// TIA Portal V18 program export: 0 tag tables, 0 data types, 83 data blocks, 120 code blocks (in call order from the OBs), 84 instance data blocks

DATA_BLOCK "GeneralDebug"   // DB1
{ S7_Optimized_Access := 'TRUE' }
// stored: MemoryReserve 100
   VAR
      Debug : Array[1..99] of Bool;
   END_VAR
BEGIN
END_DATA_BLOCK

DATA_BLOCK "DB_Commissioning"   // DB32767
{ S7_Optimized_Access := 'TRUE' }
// stored: AutoNumber false, MemoryReserve 100
   VAR RETAIN
      str : Array[1..8] of String[60];
      bit : Array[1..8] of Bool;
   END_VAR
BEGIN
   str[1] := 'LE4B171420124M33700000131950710';
END_DATA_BLOCK

DATA_BLOCK "DB_MES_Monitoring"   // DB8
{ S7_Optimized_Access := 'TRUE' }
AUTHOR : caisik - mr. machinist
// stored: MemoryReserve 100
   VAR
      Diag { S7_SetPoint := 'True'} : "UDT_MES_Monitoring";
   END_VAR
BEGIN
END_DATA_BLOCK

DATA_BLOCK "DB_ALL_PROCESS_PARAMETERS"   // DB5000
{ S7_Optimized_Access := 'TRUE' }
// stored: AutoNumber false, MemoryReserve 1000
   VAR RETAIN
      "Choosen Recipe Number" : Bool;
      ACTUAL_CHOOSEN_TYPE : "UDT_OP10_Recipe_type";   // THERE IS ASCTUAL DATA READED OUT FROM LIBRARY OF 20 TYPES BELOW
      PRODUCT_TYPE : Array[1..10] of "UDT_OP10_Recipe_type";   // PACK OF TWENTY DIFFERENT TYPES PRODUCT AND THEIR PARAMETERS FOR THE PROCESS
   END_VAR
BEGIN
   ACTUAL_CHOOSEN_TYPE.Header.RecipeName := 'produkt 1';
   ACTUAL_CHOOSEN_TYPE.Header.RecipeID := 2;
   ACTUAL_CHOOSEN_TYPE.Header."Version" := 19629;
   ACTUAL_CHOOSEN_TYPE.Header.LastModified := DTL#2026-01-17-04:23:27.501;
   ACTUAL_CHOOSEN_TYPE.Header.PartType := 'additional  name';
   ACTUAL_CHOOSEN_TYPE.Process.Timers.Delay_glue_init_start := T#2S;
   ACTUAL_CHOOSEN_TYPE.Process.Timers.Delay_Medium := T#600MS;
   ACTUAL_CHOOSEN_TYPE.Process.Timers.Delay_Long := T#2S;
   ACTUAL_CHOOSEN_TYPE.Process.Timers.Cylinder_ActTime := T#6S;
   ACTUAL_CHOOSEN_TYPE.Process.Limits.RetryLimit := 3;
   ACTUAL_CHOOSEN_TYPE.Process.Press.B1_Program := 1;
   ACTUAL_CHOOSEN_TYPE.Process.Press.B2_Program := 1;
   ACTUAL_CHOOSEN_TYPE.Process.Vision.CGlueShaftIV3_Progs[1] := 16#0001;
   ACTUAL_CHOOSEN_TYPE.Process.Vision.CGlueShaftIV3_Progs[2] := 16#0002;
   ACTUAL_CHOOSEN_TYPE.Process.Vision.CGlueShaftIV3_Progs[3] := 16#0003;
   ACTUAL_CHOOSEN_TYPE.Process.Vision.CGlueShaftIV3_Progs[4] := 16#0004;
   ACTUAL_CHOOSEN_TYPE.Process.Vision.CGlueMagnetIV3_Prog := 16#0001;
   ACTUAL_CHOOSEN_TYPE.Process.Vision.CGlueProgram := 1;
   ACTUAL_CHOOSEN_TYPE."Tooling Code".A1_Table[1] := 'SZ23055-OP010-E-Compressor-ring1 Loading tooling-1';
   ACTUAL_CHOOSEN_TYPE."Tooling Code".A1_Table[2] := 'SZ23055-OP010-E-Compressor-ring1 Loading tooling-2';
   ACTUAL_CHOOSEN_TYPE."Tooling Code".A1_Table[3] := 'SZ23055-OP010-E-Compressor-ring1 Loading tooling-3';
   ACTUAL_CHOOSEN_TYPE."Tooling Code".A1_Table[4] := 'SZ23055-OP010-E-Compressor-ring1 Loading tooling-4';
   ACTUAL_CHOOSEN_TYPE."Tooling Code".A1_Table[5] := 'SZ23055-OP010-E-Compressor-ring1 Loading tooling-5';
   ACTUAL_CHOOSEN_TYPE."Tooling Code".A1_Table[6] := 'SZ23055-OP010-E-Compressor-ring1 Loading tooling-6';
   ACTUAL_CHOOSEN_TYPE."Tooling Code".A1_Table[7] := 'SZ23055-OP010-E-Compressor-ring1 Loading tooling-7';
   ACTUAL_CHOOSEN_TYPE."Tooling Code".A1_Table[8] := 'SZ23055-OP010-E-Compressor-ring1 Loading tooling-8';
   ACTUAL_CHOOSEN_TYPE."Tooling Code".A2_Table[1] := 'SZ23055-OP010-E-Compresspr-ring1 cutting tool';
   ACTUAL_CHOOSEN_TYPE."Tooling Code".A2_Table[2] := 'SZ23055-OP010-E-Compressor-Left NG tooling-1';
   ACTUAL_CHOOSEN_TYPE."Tooling Code".A2_Table[3] := 'SZ23055-OP010-E-Compressor-shaft Rotating scanning tooling-1';
   ACTUAL_CHOOSEN_TYPE."Tooling Code".A2_Table[4] := 'SZ23055-OP010-E-Compressor-ring1 Below Positioning fixture -1';
   ACTUAL_CHOOSEN_TYPE."Tooling Code".A2_Table[5] := 'SZ23055-OP010-E-Compressor-Point adhesive tooling-1';
   ACTUAL_CHOOSEN_TYPE."Tooling Code".A2_Table[6] := 'SZ23055-OP010-E-Compressor-ring1 Upper pressing fixture-1';
   ACTUAL_CHOOSEN_TYPE."Tooling Code".A2_Table[7] := 'SZ23055-OP010-E-Compresspr-ring2 cutting tool';
   ACTUAL_CHOOSEN_TYPE."Tooling Code".A2_Table[8] := 'SZ23055-OP010-E-Compressor-Right NG tooling-1';
   ACTUAL_CHOOSEN_TYPE."Tooling Code".ROB1_Shaft_Handling_Robot.Gripper."JAW TOOLING LEFT" := 'SZ23055-OP010-E-Compressor-robot1 ring1 Left clamping jaw tooling-1';
   ACTUAL_CHOOSEN_TYPE."Tooling Code".ROB1_Shaft_Handling_Robot.Gripper."JAW TOOLING RIGHT" := 'SZ23055-OP010-E-Compressor-robot1 ring1 Right clamping jaw tooling-2';
   ACTUAL_CHOOSEN_TYPE."Tooling Code".ROB1_Shaft_Handling_Robot.Gripper."SHAFT CLAMPING LEFT" := 'SZ23055-OP010-E-Compressor-robot1 shaft Left clamping jaw tooling-1';
   ACTUAL_CHOOSEN_TYPE."Tooling Code".ROB1_Shaft_Handling_Robot.Gripper."SHAFT CLAMPING RIGHT" := 'SZ23055-OP010-E-Compressor-robot1 shaft Right clamping jaw tooling-2';
   ACTUAL_CHOOSEN_TYPE."Tooling Code".ROB2_Main_Assembly_Robot.Gripper."JAW TOOLING LEFT" := 'SZ23055-OP010-E-Compressor-robot2 shaft Right clamping jaw tooling-2';
   ACTUAL_CHOOSEN_TYPE."Tooling Code".ROB2_Main_Assembly_Robot.Gripper."JAW TOOLING RIGHT" := 'SZ23055-OP010-E-Compressor-robot2 shaft Left clamping jaw tooling-1';
   ACTUAL_CHOOSEN_TYPE."Tooling Code".ROB2_Main_Assembly_Robot.Gripper."SHAFT CLAMPING LEFT" := 'SZ23055-OP010-E-Compressor-robot2 magnet Right clamping jaw tooling-2';
   ACTUAL_CHOOSEN_TYPE."Tooling Code".ROB2_Main_Assembly_Robot.Gripper."SHAFT CLAMPING RIGHT" := 'SZ23055-OP010-E-Compressor-robot2 magnet Right clamping jaw tooling-2';
   ACTUAL_CHOOSEN_TYPE."Tooling Code".ROB3_Unloading_Robot.Gripper."JAW TOOLING LEFT" := 'SZ23055-OP010-E-Compressor-robot3 ring2 Right clamping jaw tooling-2';
   ACTUAL_CHOOSEN_TYPE."Tooling Code".ROB3_Unloading_Robot.Gripper."JAW TOOLING RIGHT" := 'SZ23055-OP010-E-Compressor-robot3 ring2 Left clamping jaw tooling-1';
   ACTUAL_CHOOSEN_TYPE."Tooling Code".ROB3_Unloading_Robot.Gripper."SHAFT CLAMPING LEFT" := 'SZ23055-OP010-E-Compressor-robot3 shaft Left clamping jaw tooling-1';
   ACTUAL_CHOOSEN_TYPE."Tooling Code".ROB3_Unloading_Robot.Gripper."SHAFT CLAMPING RIGHT" := 'SZ23055-OP010-E-Compressor-robot3 shaft Right clamping jaw tooling-2';
   ACTUAL_CHOOSEN_TYPE."Tooling Code".A1_Fixtures.A1RingUnloadingFixtureCode := 'SZ23055-OP010-E-Compresspr-ring1 cutting tool';
   ACTUAL_CHOOSEN_TYPE."Tooling Code".A1_Fixtures.E1LoadingNGFixtureCode := 'SZ23055-OP010-E-Compressor-Left NG tooling-1';
   ACTUAL_CHOOSEN_TYPE."Tooling Code".A1_Fixtures.ShaftScanFixtureCode := 'SZ23055-OP010-E-Compressor-shaft Rotating scanning tooling-1';
   ACTUAL_CHOOSEN_TYPE."Tooling Code".A1_Fixtures.B1PressFixtureCode := 'SZ23055-OP010-E-Compressor-ring1 Below Positioning fixture -1';
   ACTUAL_CHOOSEN_TYPE."Tooling Code".A1_Fixtures.CGlueFixtureCode := 'SZ23055-OP010-E-Compressor-Point adhesive tooling-1';
   ACTUAL_CHOOSEN_TYPE."Tooling Code".A1_Fixtures.B1PressCylFixtureCode := 'SZ23055-OP010-E-Compressor-ring1 Upper pressing fixture-1';
   ACTUAL_CHOOSEN_TYPE."Tooling Code".A2_Fixtures.A2RingUnloadingFixtureCode := 'SZ23055-OP010-E-Compresspr-ring2 cutting tool';
   ACTUAL_CHOOSEN_TYPE."Tooling Code".A2_Fixtures.E2UnloadingNGFixtureCode := 'SZ23055-OP010-E-Compressor-Right NG tooling-1';
   ACTUAL_CHOOSEN_TYPE."Tooling Code".A2_Fixtures.B2PressFixtureCode := 'SZ23055-OP010-E-Compressor-ring2 Below Positioning fixture -1';
   ACTUAL_CHOOSEN_TYPE."Tooling Code".A2_Fixtures.CGlueNGFixtureCode := 'SZ23055-OP010-E-Compressor-NG middle shift tooling-1';
   ACTUAL_CHOOSEN_TYPE."Tooling Code".A2_Fixtures.B2PressCylFixtureCode := 'SZ23055-OP010-E-Compressor-ring2 Upper pressing fixture-1';
   ACTUAL_CHOOSEN_TYPE.Motion.Gluing_Nozzle_Z.Position[1].Pos := 143.76;
   ACTUAL_CHOOSEN_TYPE.Motion.Gluing_Nozzle_Z.Position[2].Pos := 139.11;
   ACTUAL_CHOOSEN_TYPE.Motion.Gluing_Nozzle_Z.Position[3].Pos := 131.98;
   ACTUAL_CHOOSEN_TYPE.Motion.Gluing_Nozzle_Z.Position[4].Pos := 127.89;
   ACTUAL_CHOOSEN_TYPE.Motion.Gluing_Nozzle_Z.Position[6].Pos := 127.0;
   ACTUAL_CHOOSEN_TYPE.Motion.Gluing_Nozzle_Z.Position[7].Pos := 48.11;
   ACTUAL_CHOOSEN_TYPE.Motion.Gluing_Nozzle_Z.Position[9].Pos := 123.0;
   ACTUAL_CHOOSEN_TYPE.Motion.Gluing_Nozzle_Z.Position[1..4].Vel := 200;
   ACTUAL_CHOOSEN_TYPE.Motion.Gluing_Nozzle_Z.Position[6..9].Vel := 200;
   ACTUAL_CHOOSEN_TYPE.Motion.Gluing_Nozzle_X.Position[1].Pos := 2.34;
   ACTUAL_CHOOSEN_TYPE.Motion.Gluing_Nozzle_X.Position[2].Pos := 76.0;
   ACTUAL_CHOOSEN_TYPE.Motion.Gluing_Nozzle_X.Position[3..6].Pos := 84.69;
   ACTUAL_CHOOSEN_TYPE.Motion.Gluing_Nozzle_X.Position[7].Pos := 85.0;
   ACTUAL_CHOOSEN_TYPE.Motion.Gluing_Nozzle_X.Position[8].Pos := 88.53;
   ACTUAL_CHOOSEN_TYPE.Motion.Gluing_Nozzle_X.Position[1..8].Vel := 200;
   ACTUAL_CHOOSEN_TYPE.Motion.Gluing_Nozzle_Y.Position[1..5].Pos := 115.47;
   ACTUAL_CHOOSEN_TYPE.Motion.Gluing_Nozzle_Y.Position[6].Pos := 110.18;
   ACTUAL_CHOOSEN_TYPE.Motion.Gluing_Nozzle_Y.Position[7].Pos := 60.52;
   ACTUAL_CHOOSEN_TYPE.Motion.Gluing_Nozzle_Y.Position[8].Pos := 80.0;
   ACTUAL_CHOOSEN_TYPE.Motion.Gluing_Nozzle_Y.Position[1..7].Vel := 200;
   ACTUAL_CHOOSEN_TYPE.Motion.Gluing_Nozzle_Y.Position[8].Vel := 100;
   ACTUAL_CHOOSEN_TYPE.Motion.Ring_Turntable_Axis_1.Position[1].Pos := 3419;
   ACTUAL_CHOOSEN_TYPE.Motion.Ring_Turntable_Axis_1.Position[2].Pos := 48386;
   ACTUAL_CHOOSEN_TYPE.Motion.Ring_Turntable_Axis_1.Position[3].Pos := 93294;
   ACTUAL_CHOOSEN_TYPE.Motion.Ring_Turntable_Axis_1.Position[4].Pos := 138335;
   ACTUAL_CHOOSEN_TYPE.Motion.Ring_Turntable_Axis_1.Position[5].Pos := 183464;
   ACTUAL_CHOOSEN_TYPE.Motion.Ring_Turntable_Axis_1.Position[6].Pos := 228443;
   ACTUAL_CHOOSEN_TYPE.Motion.Ring_Turntable_Axis_1.Position[7].Pos := 273535;
   ACTUAL_CHOOSEN_TYPE.Motion.Ring_Turntable_Axis_1.Position[8].Pos := 318250;
   ACTUAL_CHOOSEN_TYPE.Motion.Ring_Turntable_Axis_1.Position[1..8].Vel := 10000;
   ACTUAL_CHOOSEN_TYPE.Motion.Shaft_Scan_Turntable_Axis.Position[2].Pos := 450000;
   ACTUAL_CHOOSEN_TYPE.Motion.Shaft_Scan_Turntable_Axis.Position[3].Pos := 900000;
   ACTUAL_CHOOSEN_TYPE.Motion.Shaft_Scan_Turntable_Axis.Position[4].Pos := 135000;
   ACTUAL_CHOOSEN_TYPE.Motion.Shaft_Scan_Turntable_Axis.Position[5].Pos := 180000;
   ACTUAL_CHOOSEN_TYPE.Motion.Shaft_Scan_Turntable_Axis.Position[6].Pos := 225000;
   ACTUAL_CHOOSEN_TYPE.Motion.Shaft_Scan_Turntable_Axis.Position[7].Pos := 270000;
   ACTUAL_CHOOSEN_TYPE.Motion.Shaft_Scan_Turntable_Axis.Position[8].Pos := 315000;
   ACTUAL_CHOOSEN_TYPE.Motion.Shaft_Scan_Turntable_Axis.Position[1..8].Vel := 10000;
   ACTUAL_CHOOSEN_TYPE.Motion.Gluing_Rotary_Jig_Axis.Position[3..6].Pos := 680000;
   ACTUAL_CHOOSEN_TYPE.Motion.Gluing_Rotary_Jig_Axis.Position[7].Pos := 90000;
   ACTUAL_CHOOSEN_TYPE.Motion.Gluing_Rotary_Jig_Axis.Position[8].Pos := 180000;
   ACTUAL_CHOOSEN_TYPE.Motion.Gluing_Rotary_Jig_Axis.Position[9].Pos := 270000;
   ACTUAL_CHOOSEN_TYPE.Motion.Gluing_Rotary_Jig_Axis.Position[1..2].Vel := 20000;
   ACTUAL_CHOOSEN_TYPE.Motion.Gluing_Rotary_Jig_Axis.Position[3..9].Vel := 10000;
   ACTUAL_CHOOSEN_TYPE.Motion.Ring_Turntable_Axis_2.Position[1].Pos := 3585;
   ACTUAL_CHOOSEN_TYPE.Motion.Ring_Turntable_Axis_2.Position[2].Pos := 48610;
   ACTUAL_CHOOSEN_TYPE.Motion.Ring_Turntable_Axis_2.Position[3].Pos := 93637;
   ACTUAL_CHOOSEN_TYPE.Motion.Ring_Turntable_Axis_2.Position[4].Pos := 138606;
   ACTUAL_CHOOSEN_TYPE.Motion.Ring_Turntable_Axis_2.Position[5].Pos := 183388;
   ACTUAL_CHOOSEN_TYPE.Motion.Ring_Turntable_Axis_2.Position[6].Pos := 228458;
   ACTUAL_CHOOSEN_TYPE.Motion.Ring_Turntable_Axis_2.Position[7].Pos := 273513;
   ACTUAL_CHOOSEN_TYPE.Motion.Ring_Turntable_Axis_2.Position[8].Pos := 318501;
   ACTUAL_CHOOSEN_TYPE.Motion.Ring_Turntable_Axis_2.Position[1..8].Vel := 10000;
   PRODUCT_TYPE[1].Header.RecipeName := 'produkt 1';
   PRODUCT_TYPE[3].Header.RecipeName := 'produkt 1';
   PRODUCT_TYPE[10].Header.RecipeName := 'produkt 1';
   PRODUCT_TYPE[1].Header.RecipeID := 1;
   PRODUCT_TYPE[3].Header.RecipeID := 1;
   PRODUCT_TYPE[10].Header.RecipeID := 1;
   PRODUCT_TYPE[1].Header."Version" := 1;
   PRODUCT_TYPE[3].Header."Version" := 1;
   PRODUCT_TYPE[10].Header."Version" := 1;
   PRODUCT_TYPE[1].Header.LastModified := DTL#2026-01-17-04:23:27.501;
   PRODUCT_TYPE[3].Header.LastModified := DTL#2026-01-17-04:23:27.501;
   PRODUCT_TYPE[10].Header.LastModified := DTL#2026-01-17-04:23:27.501;
   PRODUCT_TYPE[1].Header.PartType := 'additional  name';
   PRODUCT_TYPE[3].Header.PartType := 'additional  name';
   PRODUCT_TYPE[10].Header.PartType := 'additional  name';
   PRODUCT_TYPE[1].Process.Timers.Delay_glue_init_start := T#2S;
   PRODUCT_TYPE[2].Process.Timers.Delay_glue_init_start := T#0MS;
   PRODUCT_TYPE[3].Process.Timers.Delay_glue_init_start := T#300MS;
   PRODUCT_TYPE[4..9].Process.Timers.Delay_glue_init_start := T#0MS;
   PRODUCT_TYPE[10].Process.Timers.Delay_glue_init_start := T#2S;
   PRODUCT_TYPE[1].Process.Timers.Delay_Medium := T#600MS;
   PRODUCT_TYPE[3].Process.Timers.Delay_Medium := T#600MS;
   PRODUCT_TYPE[10].Process.Timers.Delay_Medium := T#600MS;
   PRODUCT_TYPE[1].Process.Timers.Delay_Long := T#2S;
   PRODUCT_TYPE[3].Process.Timers.Delay_Long := T#2S;
   PRODUCT_TYPE[10].Process.Timers.Delay_Long := T#2S;
   PRODUCT_TYPE[1].Process.Timers.Cylinder_ActTime := T#6S;
   PRODUCT_TYPE[3].Process.Timers.Cylinder_ActTime := T#6S;
   PRODUCT_TYPE[10].Process.Timers.Cylinder_ActTime := T#6S;
   PRODUCT_TYPE[1].Process.Limits.RetryLimit := 3;
   PRODUCT_TYPE[3].Process.Limits.RetryLimit := 3;
   PRODUCT_TYPE[10].Process.Limits.RetryLimit := 3;
   PRODUCT_TYPE[1].Process.Press.B1_Program := 1;
   PRODUCT_TYPE[3].Process.Press.B1_Program := 1;
   PRODUCT_TYPE[10].Process.Press.B1_Program := 1;
   PRODUCT_TYPE[1].Process.Press.B2_Program := 1;
   PRODUCT_TYPE[3].Process.Press.B2_Program := 1;
   PRODUCT_TYPE[10].Process.Press.B2_Program := 1;
   PRODUCT_TYPE[1].Process.Vision.CGlueShaftIV3_Progs[1] := 16#0001;
   PRODUCT_TYPE[1].Process.Vision.CGlueShaftIV3_Progs[2] := 16#0002;
   PRODUCT_TYPE[1].Process.Vision.CGlueShaftIV3_Progs[3] := 16#0003;
   PRODUCT_TYPE[1].Process.Vision.CGlueShaftIV3_Progs[4] := 16#0004;
   PRODUCT_TYPE[3].Process.Vision.CGlueShaftIV3_Progs[1] := 16#0001;
   PRODUCT_TYPE[3].Process.Vision.CGlueShaftIV3_Progs[2] := 16#0002;
   PRODUCT_TYPE[3].Process.Vision.CGlueShaftIV3_Progs[3] := 16#0003;
   PRODUCT_TYPE[3].Process.Vision.CGlueShaftIV3_Progs[4] := 16#0004;
   PRODUCT_TYPE[10].Process.Vision.CGlueShaftIV3_Progs[1] := 16#0001;
   PRODUCT_TYPE[10].Process.Vision.CGlueShaftIV3_Progs[2] := 16#0002;
   PRODUCT_TYPE[10].Process.Vision.CGlueShaftIV3_Progs[3] := 16#0003;
   PRODUCT_TYPE[10].Process.Vision.CGlueShaftIV3_Progs[4] := 16#0004;
   PRODUCT_TYPE[1].Process.Vision.CGlueMagnetIV3_Prog := 16#0001;
   PRODUCT_TYPE[3].Process.Vision.CGlueMagnetIV3_Prog := 16#0001;
   PRODUCT_TYPE[10].Process.Vision.CGlueMagnetIV3_Prog := 16#0001;
   PRODUCT_TYPE[1].Process.Vision.CGlueProgram := 1;
   PRODUCT_TYPE[3].Process.Vision.CGlueProgram := 1;
   PRODUCT_TYPE[10].Process.Vision.CGlueProgram := 1;
   PRODUCT_TYPE[1]."Tooling Code".A1_Table[1] := 'SZ23055-OP010-E-Compressor-ring1 Loading tooling-1';
   PRODUCT_TYPE[1]."Tooling Code".A1_Table[2] := 'SZ23055-OP010-E-Compressor-ring1 Loading tooling-2';
   PRODUCT_TYPE[1]."Tooling Code".A1_Table[3] := 'SZ23055-OP010-E-Compressor-ring1 Loading tooling-3';
   PRODUCT_TYPE[1]."Tooling Code".A1_Table[4] := 'SZ23055-OP010-E-Compressor-ring1 Loading tooling-4';
   PRODUCT_TYPE[1]."Tooling Code".A1_Table[5] := 'SZ23055-OP010-E-Compressor-ring1 Loading tooling-5';
   PRODUCT_TYPE[1]."Tooling Code".A1_Table[6] := 'SZ23055-OP010-E-Compressor-ring1 Loading tooling-6';
   PRODUCT_TYPE[1]."Tooling Code".A1_Table[7] := 'SZ23055-OP010-E-Compressor-ring1 Loading tooling-7';
   PRODUCT_TYPE[1]."Tooling Code".A1_Table[8] := 'SZ23055-OP010-E-Compressor-ring1 Loading tooling-8';
   PRODUCT_TYPE[3]."Tooling Code".A1_Table[1] := 'SZ23055-OP010-E-Compressor-ring1 Loading tooling-1';
   PRODUCT_TYPE[3]."Tooling Code".A1_Table[2] := 'SZ23055-OP010-E-Compressor-ring1 Loading tooling-2';
   PRODUCT_TYPE[3]."Tooling Code".A1_Table[3] := 'SZ23055-OP010-E-Compressor-ring1 Loading tooling-3';
   PRODUCT_TYPE[3]."Tooling Code".A1_Table[4] := 'SZ23055-OP010-E-Compressor-ring1 Loading tooling-4';
   PRODUCT_TYPE[3]."Tooling Code".A1_Table[5] := 'SZ23055-OP010-E-Compressor-ring1 Loading tooling-5';
   PRODUCT_TYPE[3]."Tooling Code".A1_Table[6] := 'SZ23055-OP010-E-Compressor-ring1 Loading tooling-6';
   PRODUCT_TYPE[3]."Tooling Code".A1_Table[7] := 'SZ23055-OP010-E-Compressor-ring1 Loading tooling-7';
   PRODUCT_TYPE[3]."Tooling Code".A1_Table[8] := 'SZ23055-OP010-E-Compressor-ring1 Loading tooling-8';
   PRODUCT_TYPE[10]."Tooling Code".A1_Table[1] := 'SZ23055-OP010-E-Compressor-ring1 Loading tooling-1';
   PRODUCT_TYPE[10]."Tooling Code".A1_Table[2] := 'SZ23055-OP010-E-Compressor-ring1 Loading tooling-2';
   PRODUCT_TYPE[10]."Tooling Code".A1_Table[3] := 'SZ23055-OP010-E-Compressor-ring1 Loading tooling-3';
   PRODUCT_TYPE[10]."Tooling Code".A1_Table[4] := 'SZ23055-OP010-E-Compressor-ring1 Loading tooling-4';
   PRODUCT_TYPE[10]."Tooling Code".A1_Table[5] := 'SZ23055-OP010-E-Compressor-ring1 Loading tooling-5';
   PRODUCT_TYPE[10]."Tooling Code".A1_Table[6] := 'SZ23055-OP010-E-Compressor-ring1 Loading tooling-6';
   PRODUCT_TYPE[10]."Tooling Code".A1_Table[7] := 'SZ23055-OP010-E-Compressor-ring1 Loading tooling-7';
   PRODUCT_TYPE[10]."Tooling Code".A1_Table[8] := 'SZ23055-OP010-E-Compressor-ring1 Loading tooling-8';
   PRODUCT_TYPE[1]."Tooling Code".A2_Table[1] := 'SZ23055-OP010-E-Compresspr-ring1 cutting tool';
   PRODUCT_TYPE[1]."Tooling Code".A2_Table[2] := 'SZ23055-OP010-E-Compressor-Left NG tooling-1';
   PRODUCT_TYPE[1]."Tooling Code".A2_Table[3] := 'SZ23055-OP010-E-Compressor-shaft Rotating scanning tooling-1';
   PRODUCT_TYPE[1]."Tooling Code".A2_Table[4] := 'SZ23055-OP010-E-Compressor-ring1 Below Positioning fixture -1';
   PRODUCT_TYPE[1]."Tooling Code".A2_Table[5] := 'SZ23055-OP010-E-Compressor-Point adhesive tooling-1';
   PRODUCT_TYPE[1]."Tooling Code".A2_Table[6] := 'SZ23055-OP010-E-Compressor-ring1 Upper pressing fixture-1';
   PRODUCT_TYPE[1]."Tooling Code".A2_Table[7] := 'SZ23055-OP010-E-Compresspr-ring2 cutting tool';
   PRODUCT_TYPE[1]."Tooling Code".A2_Table[8] := 'SZ23055-OP010-E-Compressor-Right NG tooling-1';
   PRODUCT_TYPE[3]."Tooling Code".A2_Table[1] := 'SZ23055-OP010-E-Compresspr-ring1 cutting tool';
   PRODUCT_TYPE[3]."Tooling Code".A2_Table[2] := 'SZ23055-OP010-E-Compressor-Left NG tooling-1';
   PRODUCT_TYPE[3]."Tooling Code".A2_Table[3] := 'SZ23055-OP010-E-Compressor-shaft Rotating scanning tooling-1';
   PRODUCT_TYPE[3]."Tooling Code".A2_Table[4] := 'SZ23055-OP010-E-Compressor-ring1 Below Positioning fixture -1';
   PRODUCT_TYPE[3]."Tooling Code".A2_Table[5] := 'SZ23055-OP010-E-Compressor-Point adhesive tooling-1';
   PRODUCT_TYPE[3]."Tooling Code".A2_Table[6] := 'SZ23055-OP010-E-Compressor-ring1 Upper pressing fixture-1';
   PRODUCT_TYPE[3]."Tooling Code".A2_Table[7] := 'SZ23055-OP010-E-Compresspr-ring2 cutting tool';
   PRODUCT_TYPE[3]."Tooling Code".A2_Table[8] := 'SZ23055-OP010-E-Compressor-Right NG tooling-1';
   PRODUCT_TYPE[10]."Tooling Code".A2_Table[1] := 'SZ23055-OP010-E-Compresspr-ring1 cutting tool';
   PRODUCT_TYPE[10]."Tooling Code".A2_Table[2] := 'SZ23055-OP010-E-Compressor-Left NG tooling-1';
   PRODUCT_TYPE[10]."Tooling Code".A2_Table[3] := 'SZ23055-OP010-E-Compressor-shaft Rotating scanning tooling-1';
   PRODUCT_TYPE[10]."Tooling Code".A2_Table[4] := 'SZ23055-OP010-E-Compressor-ring1 Below Positioning fixture -1';
   PRODUCT_TYPE[10]."Tooling Code".A2_Table[5] := 'SZ23055-OP010-E-Compressor-Point adhesive tooling-1';
   PRODUCT_TYPE[10]."Tooling Code".A2_Table[6] := 'SZ23055-OP010-E-Compressor-ring1 Upper pressing fixture-1';
   PRODUCT_TYPE[10]."Tooling Code".A2_Table[7] := 'SZ23055-OP010-E-Compresspr-ring2 cutting tool';
   PRODUCT_TYPE[10]."Tooling Code".A2_Table[8] := 'SZ23055-OP010-E-Compressor-Right NG tooling-1';
   PRODUCT_TYPE[1]."Tooling Code".ROB1_Shaft_Handling_Robot.Gripper."JAW TOOLING LEFT" := 'SZ23055-OP010-E-Compressor-robot1 ring1 Left clamping jaw tooling-1';
   PRODUCT_TYPE[3]."Tooling Code".ROB1_Shaft_Handling_Robot.Gripper."JAW TOOLING LEFT" := 'SZ23055-OP010-E-Compressor-robot1 ring1 Left clamping jaw tooling-1';
   PRODUCT_TYPE[10]."Tooling Code".ROB1_Shaft_Handling_Robot.Gripper."JAW TOOLING LEFT" := 'SZ23055-OP010-E-Compressor-robot1 ring1 Left clamping jaw tooling-1';
   PRODUCT_TYPE[1]."Tooling Code".ROB1_Shaft_Handling_Robot.Gripper."JAW TOOLING RIGHT" := 'SZ23055-OP010-E-Compressor-robot1 ring1 Right clamping jaw tooling-2';
   PRODUCT_TYPE[3]."Tooling Code".ROB1_Shaft_Handling_Robot.Gripper."JAW TOOLING RIGHT" := 'SZ23055-OP010-E-Compressor-robot1 ring1 Right clamping jaw tooling-2';
   PRODUCT_TYPE[10]."Tooling Code".ROB1_Shaft_Handling_Robot.Gripper."JAW TOOLING RIGHT" := 'SZ23055-OP010-E-Compressor-robot1 ring1 Right clamping jaw tooling-2';
   PRODUCT_TYPE[1]."Tooling Code".ROB1_Shaft_Handling_Robot.Gripper."SHAFT CLAMPING LEFT" := 'SZ23055-OP010-E-Compressor-robot1 shaft Left clamping jaw tooling-1';
   PRODUCT_TYPE[3]."Tooling Code".ROB1_Shaft_Handling_Robot.Gripper."SHAFT CLAMPING LEFT" := 'SZ23055-OP010-E-Compressor-robot1 shaft Left clamping jaw tooling-1';
   PRODUCT_TYPE[10]."Tooling Code".ROB1_Shaft_Handling_Robot.Gripper."SHAFT CLAMPING LEFT" := 'SZ23055-OP010-E-Compressor-robot1 shaft Left clamping jaw tooling-1';
   PRODUCT_TYPE[1]."Tooling Code".ROB1_Shaft_Handling_Robot.Gripper."SHAFT CLAMPING RIGHT" := 'SZ23055-OP010-E-Compressor-robot1 shaft Right clamping jaw tooling-2';
   PRODUCT_TYPE[3]."Tooling Code".ROB1_Shaft_Handling_Robot.Gripper."SHAFT CLAMPING RIGHT" := 'SZ23055-OP010-E-Compressor-robot1 shaft Right clamping jaw tooling-2';
   PRODUCT_TYPE[10]."Tooling Code".ROB1_Shaft_Handling_Robot.Gripper."SHAFT CLAMPING RIGHT" := 'SZ23055-OP010-E-Compressor-robot1 shaft Right clamping jaw tooling-2';
   PRODUCT_TYPE[1]."Tooling Code".ROB2_Main_Assembly_Robot.Gripper."JAW TOOLING LEFT" := 'SZ23055-OP010-E-Compressor-robot2 shaft Right clamping jaw tooling-2';
   PRODUCT_TYPE[3]."Tooling Code".ROB2_Main_Assembly_Robot.Gripper."JAW TOOLING LEFT" := 'SZ23055-OP010-E-Compressor-robot2 shaft Right clamping jaw tooling-2';
   PRODUCT_TYPE[10]."Tooling Code".ROB2_Main_Assembly_Robot.Gripper."JAW TOOLING LEFT" := 'SZ23055-OP010-E-Compressor-robot2 shaft Right clamping jaw tooling-2';
   PRODUCT_TYPE[1]."Tooling Code".ROB2_Main_Assembly_Robot.Gripper."JAW TOOLING RIGHT" := 'SZ23055-OP010-E-Compressor-robot2 shaft Left clamping jaw tooling-1';
   PRODUCT_TYPE[3]."Tooling Code".ROB2_Main_Assembly_Robot.Gripper."JAW TOOLING RIGHT" := 'SZ23055-OP010-E-Compressor-robot2 shaft Left clamping jaw tooling-1';
   PRODUCT_TYPE[10]."Tooling Code".ROB2_Main_Assembly_Robot.Gripper."JAW TOOLING RIGHT" := 'SZ23055-OP010-E-Compressor-robot2 shaft Left clamping jaw tooling-1';
   PRODUCT_TYPE[1]."Tooling Code".ROB2_Main_Assembly_Robot.Gripper."SHAFT CLAMPING LEFT" := 'SZ23055-OP010-E-Compressor-robot2 magnet Right clamping jaw tooling-2';
   PRODUCT_TYPE[3]."Tooling Code".ROB2_Main_Assembly_Robot.Gripper."SHAFT CLAMPING LEFT" := 'SZ23055-OP010-E-Compressor-robot2 magnet Right clamping jaw tooling-2';
   PRODUCT_TYPE[10]."Tooling Code".ROB2_Main_Assembly_Robot.Gripper."SHAFT CLAMPING LEFT" := 'SZ23055-OP010-E-Compressor-robot2 magnet Right clamping jaw tooling-2';
   PRODUCT_TYPE[1]."Tooling Code".ROB2_Main_Assembly_Robot.Gripper."SHAFT CLAMPING RIGHT" := 'SZ23055-OP010-E-Compressor-robot2 magnet Right clamping jaw tooling-2';
   PRODUCT_TYPE[3]."Tooling Code".ROB2_Main_Assembly_Robot.Gripper."SHAFT CLAMPING RIGHT" := 'SZ23055-OP010-E-Compressor-robot2 magnet Right clamping jaw tooling-2';
   PRODUCT_TYPE[10]."Tooling Code".ROB2_Main_Assembly_Robot.Gripper."SHAFT CLAMPING RIGHT" := 'SZ23055-OP010-E-Compressor-robot2 magnet Right clamping jaw tooling-2';
   PRODUCT_TYPE[1]."Tooling Code".ROB3_Unloading_Robot.Gripper."JAW TOOLING LEFT" := 'SZ23055-OP010-E-Compressor-robot3 ring2 Right clamping jaw tooling-2';
   PRODUCT_TYPE[3]."Tooling Code".ROB3_Unloading_Robot.Gripper."JAW TOOLING LEFT" := 'SZ23055-OP010-E-Compressor-robot3 ring2 Right clamping jaw tooling-2';
   PRODUCT_TYPE[10]."Tooling Code".ROB3_Unloading_Robot.Gripper."JAW TOOLING LEFT" := 'SZ23055-OP010-E-Compressor-robot3 ring2 Right clamping jaw tooling-2';
   PRODUCT_TYPE[1]."Tooling Code".ROB3_Unloading_Robot.Gripper."JAW TOOLING RIGHT" := 'SZ23055-OP010-E-Compressor-robot3 ring2 Left clamping jaw tooling-1';
   PRODUCT_TYPE[3]."Tooling Code".ROB3_Unloading_Robot.Gripper."JAW TOOLING RIGHT" := 'SZ23055-OP010-E-Compressor-robot3 ring2 Left clamping jaw tooling-1';
   PRODUCT_TYPE[10]."Tooling Code".ROB3_Unloading_Robot.Gripper."JAW TOOLING RIGHT" := 'SZ23055-OP010-E-Compressor-robot3 ring2 Left clamping jaw tooling-1';
   PRODUCT_TYPE[1]."Tooling Code".ROB3_Unloading_Robot.Gripper."SHAFT CLAMPING LEFT" := 'SZ23055-OP010-E-Compressor-robot3 shaft Left clamping jaw tooling-1';
   PRODUCT_TYPE[3]."Tooling Code".ROB3_Unloading_Robot.Gripper."SHAFT CLAMPING LEFT" := 'SZ23055-OP010-E-Compressor-robot3 shaft Left clamping jaw tooling-1';
   PRODUCT_TYPE[10]."Tooling Code".ROB3_Unloading_Robot.Gripper."SHAFT CLAMPING LEFT" := 'SZ23055-OP010-E-Compressor-robot3 shaft Left clamping jaw tooling-1';
   PRODUCT_TYPE[1]."Tooling Code".ROB3_Unloading_Robot.Gripper."SHAFT CLAMPING RIGHT" := 'SZ23055-OP010-E-Compressor-robot3 shaft Right clamping jaw tooling-2';
   PRODUCT_TYPE[3]."Tooling Code".ROB3_Unloading_Robot.Gripper."SHAFT CLAMPING RIGHT" := 'SZ23055-OP010-E-Compressor-robot3 shaft Right clamping jaw tooling-2';
   PRODUCT_TYPE[10]."Tooling Code".ROB3_Unloading_Robot.Gripper."SHAFT CLAMPING RIGHT" := 'SZ23055-OP010-E-Compressor-robot3 shaft Right clamping jaw tooling-2';
   PRODUCT_TYPE[1]."Tooling Code".A1_Fixtures.A1RingUnloadingFixtureCode := 'SZ23055-OP010-E-Compresspr-ring1 cutting tool';
   PRODUCT_TYPE[3]."Tooling Code".A1_Fixtures.A1RingUnloadingFixtureCode := 'SZ23055-OP010-E-Compresspr-ring1 cutting tool';
   PRODUCT_TYPE[10]."Tooling Code".A1_Fixtures.A1RingUnloadingFixtureCode := 'SZ23055-OP010-E-Compresspr-ring1 cutting tool';
   PRODUCT_TYPE[1]."Tooling Code".A1_Fixtures.E1LoadingNGFixtureCode := 'SZ23055-OP010-E-Compressor-Left NG tooling-1';
   PRODUCT_TYPE[3]."Tooling Code".A1_Fixtures.E1LoadingNGFixtureCode := 'SZ23055-OP010-E-Compressor-Left NG tooling-1';
   PRODUCT_TYPE[10]."Tooling Code".A1_Fixtures.E1LoadingNGFixtureCode := 'SZ23055-OP010-E-Compressor-Left NG tooling-1';
   PRODUCT_TYPE[1]."Tooling Code".A1_Fixtures.ShaftScanFixtureCode := 'SZ23055-OP010-E-Compressor-shaft Rotating scanning tooling-1';
   PRODUCT_TYPE[3]."Tooling Code".A1_Fixtures.ShaftScanFixtureCode := 'SZ23055-OP010-E-Compressor-shaft Rotating scanning tooling-1';
   PRODUCT_TYPE[10]."Tooling Code".A1_Fixtures.ShaftScanFixtureCode := 'SZ23055-OP010-E-Compressor-shaft Rotating scanning tooling-1';
   PRODUCT_TYPE[1]."Tooling Code".A1_Fixtures.B1PressFixtureCode := 'SZ23055-OP010-E-Compressor-ring1 Below Positioning fixture -1';
   PRODUCT_TYPE[3]."Tooling Code".A1_Fixtures.B1PressFixtureCode := 'SZ23055-OP010-E-Compressor-ring1 Below Positioning fixture -1';
   PRODUCT_TYPE[10]."Tooling Code".A1_Fixtures.B1PressFixtureCode := 'SZ23055-OP010-E-Compressor-ring1 Below Positioning fixture -1';
   PRODUCT_TYPE[1]."Tooling Code".A1_Fixtures.CGlueFixtureCode := 'SZ23055-OP010-E-Compressor-Point adhesive tooling-1';
   PRODUCT_TYPE[3]."Tooling Code".A1_Fixtures.CGlueFixtureCode := 'SZ23055-OP010-E-Compressor-Point adhesive tooling-1';
   PRODUCT_TYPE[10]."Tooling Code".A1_Fixtures.CGlueFixtureCode := 'SZ23055-OP010-E-Compressor-Point adhesive tooling-1';
   PRODUCT_TYPE[1]."Tooling Code".A1_Fixtures.B1PressCylFixtureCode := 'SZ23055-OP010-E-Compressor-ring1 Upper pressing fixture-1';
   PRODUCT_TYPE[3]."Tooling Code".A1_Fixtures.B1PressCylFixtureCode := 'SZ23055-OP010-E-Compressor-ring1 Upper pressing fixture-1';
   PRODUCT_TYPE[10]."Tooling Code".A1_Fixtures.B1PressCylFixtureCode := 'SZ23055-OP010-E-Compressor-ring1 Upper pressing fixture-1';
   PRODUCT_TYPE[1]."Tooling Code".A2_Fixtures.A2RingUnloadingFixtureCode := 'SZ23055-OP010-E-Compresspr-ring2 cutting tool';
   PRODUCT_TYPE[3]."Tooling Code".A2_Fixtures.A2RingUnloadingFixtureCode := 'SZ23055-OP010-E-Compresspr-ring2 cutting tool';
   PRODUCT_TYPE[10]."Tooling Code".A2_Fixtures.A2RingUnloadingFixtureCode := 'SZ23055-OP010-E-Compresspr-ring2 cutting tool';
   PRODUCT_TYPE[1]."Tooling Code".A2_Fixtures.E2UnloadingNGFixtureCode := 'SZ23055-OP010-E-Compressor-Right NG tooling-1';
   PRODUCT_TYPE[3]."Tooling Code".A2_Fixtures.E2UnloadingNGFixtureCode := 'SZ23055-OP010-E-Compressor-Right NG tooling-1';
   PRODUCT_TYPE[10]."Tooling Code".A2_Fixtures.E2UnloadingNGFixtureCode := 'SZ23055-OP010-E-Compressor-Right NG tooling-1';
   PRODUCT_TYPE[1]."Tooling Code".A2_Fixtures.B2PressFixtureCode := 'SZ23055-OP010-E-Compressor-ring2 Below Positioning fixture -1';
   PRODUCT_TYPE[3]."Tooling Code".A2_Fixtures.B2PressFixtureCode := 'SZ23055-OP010-E-Compressor-ring2 Below Positioning fixture -1';
   PRODUCT_TYPE[10]."Tooling Code".A2_Fixtures.B2PressFixtureCode := 'SZ23055-OP010-E-Compressor-ring2 Below Positioning fixture -1';
   PRODUCT_TYPE[1]."Tooling Code".A2_Fixtures.CGlueNGFixtureCode := 'SZ23055-OP010-E-Compressor-NG middle shift tooling-1';
   PRODUCT_TYPE[3]."Tooling Code".A2_Fixtures.CGlueNGFixtureCode := 'SZ23055-OP010-E-Compressor-NG middle shift tooling-1';
   PRODUCT_TYPE[10]."Tooling Code".A2_Fixtures.CGlueNGFixtureCode := 'SZ23055-OP010-E-Compressor-NG middle shift tooling-1';
   PRODUCT_TYPE[1]."Tooling Code".A2_Fixtures.B2PressCylFixtureCode := 'SZ23055-OP010-E-Compressor-ring2 Upper pressing fixture-1';
   PRODUCT_TYPE[3]."Tooling Code".A2_Fixtures.B2PressCylFixtureCode := 'SZ23055-OP010-E-Compressor-ring2 Upper pressing fixture-1';
   PRODUCT_TYPE[10]."Tooling Code".A2_Fixtures.B2PressCylFixtureCode := 'SZ23055-OP010-E-Compressor-ring2 Upper pressing fixture-1';
   PRODUCT_TYPE[1].Motion.Gluing_Nozzle_Z.Position[1].Pos := 143.76;
   PRODUCT_TYPE[1].Motion.Gluing_Nozzle_Z.Position[2].Pos := 139.11;
   PRODUCT_TYPE[1].Motion.Gluing_Nozzle_Z.Position[3].Pos := 131.98;
   PRODUCT_TYPE[1].Motion.Gluing_Nozzle_Z.Position[4].Pos := 127.89;
   PRODUCT_TYPE[1].Motion.Gluing_Nozzle_Z.Position[6].Pos := 127.0;
   PRODUCT_TYPE[1].Motion.Gluing_Nozzle_Z.Position[7].Pos := 48.11;
   PRODUCT_TYPE[1].Motion.Gluing_Nozzle_Z.Position[9].Pos := 123.0;
   PRODUCT_TYPE[2].Motion.Gluing_Nozzle_Z.Position[1].Pos := 143.76;
   PRODUCT_TYPE[2].Motion.Gluing_Nozzle_Z.Position[2].Pos := 139.11;
   PRODUCT_TYPE[2].Motion.Gluing_Nozzle_Z.Position[3].Pos := 131.98;
   PRODUCT_TYPE[2].Motion.Gluing_Nozzle_Z.Position[4].Pos := 127.89;
   PRODUCT_TYPE[2].Motion.Gluing_Nozzle_Z.Position[6].Pos := 127.0;
   PRODUCT_TYPE[2].Motion.Gluing_Nozzle_Z.Position[7].Pos := 48.11;
   PRODUCT_TYPE[2].Motion.Gluing_Nozzle_Z.Position[9].Pos := 123.0;
   PRODUCT_TYPE[3].Motion.Gluing_Nozzle_Z.Position[1].Pos := 143.76;
   PRODUCT_TYPE[3].Motion.Gluing_Nozzle_Z.Position[2].Pos := 139.11;
   PRODUCT_TYPE[3].Motion.Gluing_Nozzle_Z.Position[3].Pos := 131.98;
   PRODUCT_TYPE[3].Motion.Gluing_Nozzle_Z.Position[4].Pos := 127.89;
   PRODUCT_TYPE[3].Motion.Gluing_Nozzle_Z.Position[6].Pos := 127.0;
   PRODUCT_TYPE[3].Motion.Gluing_Nozzle_Z.Position[7].Pos := 48.11;
   PRODUCT_TYPE[3].Motion.Gluing_Nozzle_Z.Position[9].Pos := 123.0;
   PRODUCT_TYPE[4].Motion.Gluing_Nozzle_Z.Position[1].Pos := 143.76;
   PRODUCT_TYPE[4].Motion.Gluing_Nozzle_Z.Position[2].Pos := 139.11;
   PRODUCT_TYPE[4].Motion.Gluing_Nozzle_Z.Position[3].Pos := 131.98;
   PRODUCT_TYPE[4].Motion.Gluing_Nozzle_Z.Position[4].Pos := 127.89;
   PRODUCT_TYPE[4].Motion.Gluing_Nozzle_Z.Position[6].Pos := 127.0;
   PRODUCT_TYPE[4].Motion.Gluing_Nozzle_Z.Position[7].Pos := 48.11;
   PRODUCT_TYPE[4].Motion.Gluing_Nozzle_Z.Position[9].Pos := 123.0;
   PRODUCT_TYPE[5].Motion.Gluing_Nozzle_Z.Position[1].Pos := 143.76;
   PRODUCT_TYPE[5].Motion.Gluing_Nozzle_Z.Position[2].Pos := 139.11;
   PRODUCT_TYPE[5].Motion.Gluing_Nozzle_Z.Position[3].Pos := 131.98;
   PRODUCT_TYPE[5].Motion.Gluing_Nozzle_Z.Position[4].Pos := 127.89;
   PRODUCT_TYPE[5].Motion.Gluing_Nozzle_Z.Position[6].Pos := 127.0;
   PRODUCT_TYPE[5].Motion.Gluing_Nozzle_Z.Position[7].Pos := 48.11;
   PRODUCT_TYPE[5].Motion.Gluing_Nozzle_Z.Position[9].Pos := 123.0;
   PRODUCT_TYPE[6].Motion.Gluing_Nozzle_Z.Position[1].Pos := 143.76;
   PRODUCT_TYPE[6].Motion.Gluing_Nozzle_Z.Position[2].Pos := 139.11;
   PRODUCT_TYPE[6].Motion.Gluing_Nozzle_Z.Position[3].Pos := 131.98;
   PRODUCT_TYPE[6].Motion.Gluing_Nozzle_Z.Position[4].Pos := 127.89;
   PRODUCT_TYPE[6].Motion.Gluing_Nozzle_Z.Position[6].Pos := 127.0;
   PRODUCT_TYPE[6].Motion.Gluing_Nozzle_Z.Position[7].Pos := 48.11;
   PRODUCT_TYPE[6].Motion.Gluing_Nozzle_Z.Position[9].Pos := 123.0;
   PRODUCT_TYPE[7].Motion.Gluing_Nozzle_Z.Position[1].Pos := 143.76;
   PRODUCT_TYPE[7].Motion.Gluing_Nozzle_Z.Position[2].Pos := 139.11;
   PRODUCT_TYPE[7].Motion.Gluing_Nozzle_Z.Position[3].Pos := 131.98;
   PRODUCT_TYPE[7].Motion.Gluing_Nozzle_Z.Position[4].Pos := 127.89;
   PRODUCT_TYPE[7].Motion.Gluing_Nozzle_Z.Position[6].Pos := 127.0;
   PRODUCT_TYPE[7].Motion.Gluing_Nozzle_Z.Position[7].Pos := 48.11;
   PRODUCT_TYPE[7].Motion.Gluing_Nozzle_Z.Position[9].Pos := 123.0;
   PRODUCT_TYPE[8].Motion.Gluing_Nozzle_Z.Position[1].Pos := 143.76;
   PRODUCT_TYPE[8].Motion.Gluing_Nozzle_Z.Position[2].Pos := 139.11;
   PRODUCT_TYPE[8].Motion.Gluing_Nozzle_Z.Position[3].Pos := 131.98;
   PRODUCT_TYPE[8].Motion.Gluing_Nozzle_Z.Position[4].Pos := 127.89;
   PRODUCT_TYPE[8].Motion.Gluing_Nozzle_Z.Position[6].Pos := 127.0;
   PRODUCT_TYPE[8].Motion.Gluing_Nozzle_Z.Position[7].Pos := 48.11;
   PRODUCT_TYPE[8].Motion.Gluing_Nozzle_Z.Position[9].Pos := 123.0;
   PRODUCT_TYPE[9].Motion.Gluing_Nozzle_Z.Position[1].Pos := 143.76;
   PRODUCT_TYPE[9].Motion.Gluing_Nozzle_Z.Position[2].Pos := 139.11;
   PRODUCT_TYPE[9].Motion.Gluing_Nozzle_Z.Position[3].Pos := 131.98;
   PRODUCT_TYPE[9].Motion.Gluing_Nozzle_Z.Position[4].Pos := 127.89;
   PRODUCT_TYPE[9].Motion.Gluing_Nozzle_Z.Position[6].Pos := 127.0;
   PRODUCT_TYPE[9].Motion.Gluing_Nozzle_Z.Position[7].Pos := 48.11;
   PRODUCT_TYPE[9].Motion.Gluing_Nozzle_Z.Position[9].Pos := 123.0;
   PRODUCT_TYPE[10].Motion.Gluing_Nozzle_Z.Position[1].Pos := 143.76;
   PRODUCT_TYPE[10].Motion.Gluing_Nozzle_Z.Position[2].Pos := 139.11;
   PRODUCT_TYPE[10].Motion.Gluing_Nozzle_Z.Position[3].Pos := 131.98;
   PRODUCT_TYPE[10].Motion.Gluing_Nozzle_Z.Position[4].Pos := 127.89;
   PRODUCT_TYPE[10].Motion.Gluing_Nozzle_Z.Position[6].Pos := 127.0;
   PRODUCT_TYPE[10].Motion.Gluing_Nozzle_Z.Position[7].Pos := 48.11;
   PRODUCT_TYPE[10].Motion.Gluing_Nozzle_Z.Position[9].Pos := 123.0;
   PRODUCT_TYPE[1].Motion.Gluing_Nozzle_Z.Position[1..4].Vel := 200;
   PRODUCT_TYPE[1].Motion.Gluing_Nozzle_Z.Position[6..9].Vel := 200;
   PRODUCT_TYPE[2].Motion.Gluing_Nozzle_Z.Position[1..4].Vel := 200;
   PRODUCT_TYPE[2].Motion.Gluing_Nozzle_Z.Position[6..9].Vel := 200;
   PRODUCT_TYPE[3].Motion.Gluing_Nozzle_Z.Position[1..4].Vel := 200;
   PRODUCT_TYPE[3].Motion.Gluing_Nozzle_Z.Position[6..9].Vel := 200;
   PRODUCT_TYPE[4].Motion.Gluing_Nozzle_Z.Position[1..4].Vel := 200;
   PRODUCT_TYPE[4].Motion.Gluing_Nozzle_Z.Position[6..9].Vel := 200;
   PRODUCT_TYPE[5].Motion.Gluing_Nozzle_Z.Position[1..4].Vel := 200;
   PRODUCT_TYPE[5].Motion.Gluing_Nozzle_Z.Position[6..9].Vel := 200;
   PRODUCT_TYPE[6].Motion.Gluing_Nozzle_Z.Position[1..4].Vel := 200;
   PRODUCT_TYPE[6].Motion.Gluing_Nozzle_Z.Position[6..9].Vel := 200;
   PRODUCT_TYPE[7].Motion.Gluing_Nozzle_Z.Position[1..4].Vel := 200;
   PRODUCT_TYPE[7].Motion.Gluing_Nozzle_Z.Position[6..9].Vel := 200;
   PRODUCT_TYPE[8].Motion.Gluing_Nozzle_Z.Position[1..4].Vel := 200;
   PRODUCT_TYPE[8].Motion.Gluing_Nozzle_Z.Position[6..9].Vel := 200;
   PRODUCT_TYPE[9].Motion.Gluing_Nozzle_Z.Position[1..4].Vel := 200;
   PRODUCT_TYPE[9].Motion.Gluing_Nozzle_Z.Position[6..9].Vel := 200;
   PRODUCT_TYPE[10].Motion.Gluing_Nozzle_Z.Position[1..4].Vel := 200;
   PRODUCT_TYPE[10].Motion.Gluing_Nozzle_Z.Position[6..9].Vel := 200;
   PRODUCT_TYPE[1].Motion.Gluing_Nozzle_X.Position[1].Pos := 2.34;
   PRODUCT_TYPE[1].Motion.Gluing_Nozzle_X.Position[2].Pos := 76.0;
   PRODUCT_TYPE[1].Motion.Gluing_Nozzle_X.Position[3..6].Pos := 84.69;
   PRODUCT_TYPE[1].Motion.Gluing_Nozzle_X.Position[7].Pos := 85.0;
   PRODUCT_TYPE[1].Motion.Gluing_Nozzle_X.Position[8].Pos := 88.53;
   PRODUCT_TYPE[2].Motion.Gluing_Nozzle_X.Position[1].Pos := 2.34;
   PRODUCT_TYPE[2].Motion.Gluing_Nozzle_X.Position[2].Pos := 76.0;
   PRODUCT_TYPE[2].Motion.Gluing_Nozzle_X.Position[3..6].Pos := 84.69;
   PRODUCT_TYPE[2].Motion.Gluing_Nozzle_X.Position[7].Pos := 85.0;
   PRODUCT_TYPE[2].Motion.Gluing_Nozzle_X.Position[8].Pos := 88.53;
   PRODUCT_TYPE[3].Motion.Gluing_Nozzle_X.Position[1].Pos := 2.34;
   PRODUCT_TYPE[3].Motion.Gluing_Nozzle_X.Position[2].Pos := 76.0;
   PRODUCT_TYPE[3].Motion.Gluing_Nozzle_X.Position[3..6].Pos := 84.69;
   PRODUCT_TYPE[3].Motion.Gluing_Nozzle_X.Position[7].Pos := 85.0;
   PRODUCT_TYPE[3].Motion.Gluing_Nozzle_X.Position[8].Pos := 88.53;
   PRODUCT_TYPE[4].Motion.Gluing_Nozzle_X.Position[1].Pos := 2.34;
   PRODUCT_TYPE[4].Motion.Gluing_Nozzle_X.Position[2].Pos := 76.0;
   PRODUCT_TYPE[4].Motion.Gluing_Nozzle_X.Position[3..6].Pos := 84.69;
   PRODUCT_TYPE[4].Motion.Gluing_Nozzle_X.Position[7].Pos := 85.0;
   PRODUCT_TYPE[4].Motion.Gluing_Nozzle_X.Position[8].Pos := 88.53;
   PRODUCT_TYPE[5].Motion.Gluing_Nozzle_X.Position[1].Pos := 2.34;
   PRODUCT_TYPE[5].Motion.Gluing_Nozzle_X.Position[2].Pos := 76.0;
   PRODUCT_TYPE[5].Motion.Gluing_Nozzle_X.Position[3..6].Pos := 84.69;
   PRODUCT_TYPE[5].Motion.Gluing_Nozzle_X.Position[7].Pos := 85.0;
   PRODUCT_TYPE[5].Motion.Gluing_Nozzle_X.Position[8].Pos := 88.53;
   PRODUCT_TYPE[6].Motion.Gluing_Nozzle_X.Position[1].Pos := 2.34;
   PRODUCT_TYPE[6].Motion.Gluing_Nozzle_X.Position[2].Pos := 76.0;
   PRODUCT_TYPE[6].Motion.Gluing_Nozzle_X.Position[3..6].Pos := 84.69;
   PRODUCT_TYPE[6].Motion.Gluing_Nozzle_X.Position[7].Pos := 85.0;
   PRODUCT_TYPE[6].Motion.Gluing_Nozzle_X.Position[8].Pos := 88.53;
   PRODUCT_TYPE[7].Motion.Gluing_Nozzle_X.Position[1].Pos := 2.34;
   PRODUCT_TYPE[7].Motion.Gluing_Nozzle_X.Position[2].Pos := 76.0;
   PRODUCT_TYPE[7].Motion.Gluing_Nozzle_X.Position[3..6].Pos := 84.69;
   PRODUCT_TYPE[7].Motion.Gluing_Nozzle_X.Position[7].Pos := 85.0;
   PRODUCT_TYPE[7].Motion.Gluing_Nozzle_X.Position[8].Pos := 88.53;
   PRODUCT_TYPE[8].Motion.Gluing_Nozzle_X.Position[1].Pos := 2.34;
   PRODUCT_TYPE[8].Motion.Gluing_Nozzle_X.Position[2].Pos := 76.0;
   PRODUCT_TYPE[8].Motion.Gluing_Nozzle_X.Position[3..6].Pos := 84.69;
   PRODUCT_TYPE[8].Motion.Gluing_Nozzle_X.Position[7].Pos := 85.0;
   PRODUCT_TYPE[8].Motion.Gluing_Nozzle_X.Position[8].Pos := 88.53;
   PRODUCT_TYPE[9].Motion.Gluing_Nozzle_X.Position[1].Pos := 2.34;
   PRODUCT_TYPE[9].Motion.Gluing_Nozzle_X.Position[2].Pos := 76.0;
   PRODUCT_TYPE[9].Motion.Gluing_Nozzle_X.Position[3..6].Pos := 84.69;
   PRODUCT_TYPE[9].Motion.Gluing_Nozzle_X.Position[7].Pos := 85.0;
   PRODUCT_TYPE[9].Motion.Gluing_Nozzle_X.Position[8].Pos := 88.53;
   PRODUCT_TYPE[10].Motion.Gluing_Nozzle_X.Position[1].Pos := 2.34;
   PRODUCT_TYPE[10].Motion.Gluing_Nozzle_X.Position[2].Pos := 76.0;
   PRODUCT_TYPE[10].Motion.Gluing_Nozzle_X.Position[3..6].Pos := 84.69;
   PRODUCT_TYPE[10].Motion.Gluing_Nozzle_X.Position[7].Pos := 85.0;
   PRODUCT_TYPE[10].Motion.Gluing_Nozzle_X.Position[8].Pos := 88.53;
   PRODUCT_TYPE[1].Motion.Gluing_Nozzle_X.Position[1..8].Vel := 200;
   PRODUCT_TYPE[2].Motion.Gluing_Nozzle_X.Position[1..8].Vel := 200;
   PRODUCT_TYPE[3].Motion.Gluing_Nozzle_X.Position[1..8].Vel := 200;
   PRODUCT_TYPE[4].Motion.Gluing_Nozzle_X.Position[1..8].Vel := 200;
   PRODUCT_TYPE[5].Motion.Gluing_Nozzle_X.Position[1..8].Vel := 200;
   PRODUCT_TYPE[6].Motion.Gluing_Nozzle_X.Position[1..8].Vel := 200;
   PRODUCT_TYPE[7].Motion.Gluing_Nozzle_X.Position[1..8].Vel := 200;
   PRODUCT_TYPE[8].Motion.Gluing_Nozzle_X.Position[1..8].Vel := 200;
   PRODUCT_TYPE[9].Motion.Gluing_Nozzle_X.Position[1..8].Vel := 200;
   PRODUCT_TYPE[10].Motion.Gluing_Nozzle_X.Position[1..8].Vel := 200;
   PRODUCT_TYPE[1].Motion.Gluing_Nozzle_Y.Position[1..5].Pos := 115.47;
   PRODUCT_TYPE[1].Motion.Gluing_Nozzle_Y.Position[6].Pos := 110.18;
   PRODUCT_TYPE[1].Motion.Gluing_Nozzle_Y.Position[7].Pos := 60.52;
   PRODUCT_TYPE[1].Motion.Gluing_Nozzle_Y.Position[8].Pos := 80.0;
   PRODUCT_TYPE[2].Motion.Gluing_Nozzle_Y.Position[1..5].Pos := 115.47;
   PRODUCT_TYPE[2].Motion.Gluing_Nozzle_Y.Position[6].Pos := 110.18;
   PRODUCT_TYPE[2].Motion.Gluing_Nozzle_Y.Position[7].Pos := 60.52;
   PRODUCT_TYPE[2].Motion.Gluing_Nozzle_Y.Position[8].Pos := 80.0;
   PRODUCT_TYPE[3].Motion.Gluing_Nozzle_Y.Position[1..5].Pos := 115.47;
   PRODUCT_TYPE[3].Motion.Gluing_Nozzle_Y.Position[6].Pos := 110.18;
   PRODUCT_TYPE[3].Motion.Gluing_Nozzle_Y.Position[7].Pos := 60.52;
   PRODUCT_TYPE[3].Motion.Gluing_Nozzle_Y.Position[8].Pos := 80.0;
   PRODUCT_TYPE[4].Motion.Gluing_Nozzle_Y.Position[1..5].Pos := 115.47;
   PRODUCT_TYPE[4].Motion.Gluing_Nozzle_Y.Position[6].Pos := 110.18;
   PRODUCT_TYPE[4].Motion.Gluing_Nozzle_Y.Position[7].Pos := 60.52;
   PRODUCT_TYPE[4].Motion.Gluing_Nozzle_Y.Position[8].Pos := 80.0;
   PRODUCT_TYPE[5].Motion.Gluing_Nozzle_Y.Position[1..5].Pos := 115.47;
   PRODUCT_TYPE[5].Motion.Gluing_Nozzle_Y.Position[6].Pos := 110.18;
   PRODUCT_TYPE[5].Motion.Gluing_Nozzle_Y.Position[7].Pos := 60.52;
   PRODUCT_TYPE[5].Motion.Gluing_Nozzle_Y.Position[8].Pos := 80.0;
   PRODUCT_TYPE[6].Motion.Gluing_Nozzle_Y.Position[1..5].Pos := 115.47;
   PRODUCT_TYPE[6].Motion.Gluing_Nozzle_Y.Position[6].Pos := 110.18;
   PRODUCT_TYPE[6].Motion.Gluing_Nozzle_Y.Position[7].Pos := 60.52;
   PRODUCT_TYPE[6].Motion.Gluing_Nozzle_Y.Position[8].Pos := 80.0;
   PRODUCT_TYPE[7].Motion.Gluing_Nozzle_Y.Position[1..5].Pos := 115.47;
   PRODUCT_TYPE[7].Motion.Gluing_Nozzle_Y.Position[6].Pos := 110.18;
   PRODUCT_TYPE[7].Motion.Gluing_Nozzle_Y.Position[7].Pos := 60.52;
   PRODUCT_TYPE[7].Motion.Gluing_Nozzle_Y.Position[8].Pos := 80.0;
   PRODUCT_TYPE[8].Motion.Gluing_Nozzle_Y.Position[1..5].Pos := 115.47;
   PRODUCT_TYPE[8].Motion.Gluing_Nozzle_Y.Position[6].Pos := 110.18;
   PRODUCT_TYPE[8].Motion.Gluing_Nozzle_Y.Position[7].Pos := 60.52;
   PRODUCT_TYPE[8].Motion.Gluing_Nozzle_Y.Position[8].Pos := 80.0;
   PRODUCT_TYPE[9].Motion.Gluing_Nozzle_Y.Position[1..5].Pos := 115.47;
   PRODUCT_TYPE[9].Motion.Gluing_Nozzle_Y.Position[6].Pos := 110.18;
   PRODUCT_TYPE[9].Motion.Gluing_Nozzle_Y.Position[7].Pos := 60.52;
   PRODUCT_TYPE[9].Motion.Gluing_Nozzle_Y.Position[8].Pos := 80.0;
   PRODUCT_TYPE[10].Motion.Gluing_Nozzle_Y.Position[1..5].Pos := 115.47;
   PRODUCT_TYPE[10].Motion.Gluing_Nozzle_Y.Position[6].Pos := 110.18;
   PRODUCT_TYPE[10].Motion.Gluing_Nozzle_Y.Position[7].Pos := 60.52;
   PRODUCT_TYPE[10].Motion.Gluing_Nozzle_Y.Position[8].Pos := 80.0;
   PRODUCT_TYPE[1].Motion.Gluing_Nozzle_Y.Position[1..7].Vel := 200;
   PRODUCT_TYPE[1].Motion.Gluing_Nozzle_Y.Position[8].Vel := 100;
   PRODUCT_TYPE[2].Motion.Gluing_Nozzle_Y.Position[1..7].Vel := 200;
   PRODUCT_TYPE[2].Motion.Gluing_Nozzle_Y.Position[8].Vel := 100;
   PRODUCT_TYPE[3].Motion.Gluing_Nozzle_Y.Position[1..7].Vel := 200;
   PRODUCT_TYPE[3].Motion.Gluing_Nozzle_Y.Position[8].Vel := 100;
   PRODUCT_TYPE[4].Motion.Gluing_Nozzle_Y.Position[1..7].Vel := 200;
   PRODUCT_TYPE[4].Motion.Gluing_Nozzle_Y.Position[8].Vel := 100;
   PRODUCT_TYPE[5].Motion.Gluing_Nozzle_Y.Position[1..7].Vel := 200;
   PRODUCT_TYPE[5].Motion.Gluing_Nozzle_Y.Position[8].Vel := 100;
   PRODUCT_TYPE[6].Motion.Gluing_Nozzle_Y.Position[1..7].Vel := 200;
   PRODUCT_TYPE[6].Motion.Gluing_Nozzle_Y.Position[8].Vel := 100;
   PRODUCT_TYPE[7].Motion.Gluing_Nozzle_Y.Position[1..7].Vel := 200;
   PRODUCT_TYPE[7].Motion.Gluing_Nozzle_Y.Position[8].Vel := 100;
   PRODUCT_TYPE[8].Motion.Gluing_Nozzle_Y.Position[1..7].Vel := 200;
   PRODUCT_TYPE[8].Motion.Gluing_Nozzle_Y.Position[8].Vel := 100;
   PRODUCT_TYPE[9].Motion.Gluing_Nozzle_Y.Position[1..7].Vel := 200;
   PRODUCT_TYPE[9].Motion.Gluing_Nozzle_Y.Position[8].Vel := 100;
   PRODUCT_TYPE[10].Motion.Gluing_Nozzle_Y.Position[1..7].Vel := 200;
   PRODUCT_TYPE[10].Motion.Gluing_Nozzle_Y.Position[8].Vel := 100;
   PRODUCT_TYPE[1].Motion.Ring_Turntable_Axis_1.Position[1].Pos := 3419;
   PRODUCT_TYPE[1].Motion.Ring_Turntable_Axis_1.Position[2].Pos := 48386;
   PRODUCT_TYPE[1].Motion.Ring_Turntable_Axis_1.Position[3].Pos := 93294;
   PRODUCT_TYPE[1].Motion.Ring_Turntable_Axis_1.Position[4].Pos := 138335;
   PRODUCT_TYPE[1].Motion.Ring_Turntable_Axis_1.Position[5].Pos := 183464;
   PRODUCT_TYPE[1].Motion.Ring_Turntable_Axis_1.Position[6].Pos := 228443;
   PRODUCT_TYPE[1].Motion.Ring_Turntable_Axis_1.Position[7].Pos := 273535;
   PRODUCT_TYPE[1].Motion.Ring_Turntable_Axis_1.Position[8].Pos := 318250;
   PRODUCT_TYPE[2].Motion.Ring_Turntable_Axis_1.Position[1].Pos := 3419;
   PRODUCT_TYPE[2].Motion.Ring_Turntable_Axis_1.Position[2].Pos := 48386;
   PRODUCT_TYPE[2].Motion.Ring_Turntable_Axis_1.Position[3].Pos := 93294;
   PRODUCT_TYPE[2].Motion.Ring_Turntable_Axis_1.Position[4].Pos := 138335;
   PRODUCT_TYPE[2].Motion.Ring_Turntable_Axis_1.Position[5].Pos := 183464;
   PRODUCT_TYPE[2].Motion.Ring_Turntable_Axis_1.Position[6].Pos := 228443;
   PRODUCT_TYPE[2].Motion.Ring_Turntable_Axis_1.Position[7].Pos := 273535;
   PRODUCT_TYPE[2].Motion.Ring_Turntable_Axis_1.Position[8].Pos := 318250;
   PRODUCT_TYPE[3].Motion.Ring_Turntable_Axis_1.Position[1].Pos := 3419;
   PRODUCT_TYPE[3].Motion.Ring_Turntable_Axis_1.Position[2].Pos := 48386;
   PRODUCT_TYPE[3].Motion.Ring_Turntable_Axis_1.Position[3].Pos := 93294;
   PRODUCT_TYPE[3].Motion.Ring_Turntable_Axis_1.Position[4].Pos := 138335;
   PRODUCT_TYPE[3].Motion.Ring_Turntable_Axis_1.Position[5].Pos := 183464;
   PRODUCT_TYPE[3].Motion.Ring_Turntable_Axis_1.Position[6].Pos := 228443;
   PRODUCT_TYPE[3].Motion.Ring_Turntable_Axis_1.Position[7].Pos := 273535;
   PRODUCT_TYPE[3].Motion.Ring_Turntable_Axis_1.Position[8].Pos := 318250;
   PRODUCT_TYPE[4].Motion.Ring_Turntable_Axis_1.Position[1].Pos := 3419;
   PRODUCT_TYPE[4].Motion.Ring_Turntable_Axis_1.Position[2].Pos := 48386;
   PRODUCT_TYPE[4].Motion.Ring_Turntable_Axis_1.Position[3].Pos := 93294;
   PRODUCT_TYPE[4].Motion.Ring_Turntable_Axis_1.Position[4].Pos := 138335;
   PRODUCT_TYPE[4].Motion.Ring_Turntable_Axis_1.Position[5].Pos := 183464;
   PRODUCT_TYPE[4].Motion.Ring_Turntable_Axis_1.Position[6].Pos := 228443;
   PRODUCT_TYPE[4].Motion.Ring_Turntable_Axis_1.Position[7].Pos := 273535;
   PRODUCT_TYPE[4].Motion.Ring_Turntable_Axis_1.Position[8].Pos := 318250;
   PRODUCT_TYPE[5].Motion.Ring_Turntable_Axis_1.Position[1].Pos := 3419;
   PRODUCT_TYPE[5].Motion.Ring_Turntable_Axis_1.Position[2].Pos := 48386;
   PRODUCT_TYPE[5].Motion.Ring_Turntable_Axis_1.Position[3].Pos := 93294;
   PRODUCT_TYPE[5].Motion.Ring_Turntable_Axis_1.Position[4].Pos := 138335;
   PRODUCT_TYPE[5].Motion.Ring_Turntable_Axis_1.Position[5].Pos := 183464;
   PRODUCT_TYPE[5].Motion.Ring_Turntable_Axis_1.Position[6].Pos := 228443;
   PRODUCT_TYPE[5].Motion.Ring_Turntable_Axis_1.Position[7].Pos := 273535;
   PRODUCT_TYPE[5].Motion.Ring_Turntable_Axis_1.Position[8].Pos := 318250;
   PRODUCT_TYPE[6].Motion.Ring_Turntable_Axis_1.Position[1].Pos := 3419;
   PRODUCT_TYPE[6].Motion.Ring_Turntable_Axis_1.Position[2].Pos := 48386;
   PRODUCT_TYPE[6].Motion.Ring_Turntable_Axis_1.Position[3].Pos := 93294;
   PRODUCT_TYPE[6].Motion.Ring_Turntable_Axis_1.Position[4].Pos := 138335;
   PRODUCT_TYPE[6].Motion.Ring_Turntable_Axis_1.Position[5].Pos := 183464;
   PRODUCT_TYPE[6].Motion.Ring_Turntable_Axis_1.Position[6].Pos := 228443;
   PRODUCT_TYPE[6].Motion.Ring_Turntable_Axis_1.Position[7].Pos := 273535;
   PRODUCT_TYPE[6].Motion.Ring_Turntable_Axis_1.Position[8].Pos := 318250;
   PRODUCT_TYPE[7].Motion.Ring_Turntable_Axis_1.Position[1].Pos := 3419;
   PRODUCT_TYPE[7].Motion.Ring_Turntable_Axis_1.Position[2].Pos := 48386;
   PRODUCT_TYPE[7].Motion.Ring_Turntable_Axis_1.Position[3].Pos := 93294;
   PRODUCT_TYPE[7].Motion.Ring_Turntable_Axis_1.Position[4].Pos := 138335;
   PRODUCT_TYPE[7].Motion.Ring_Turntable_Axis_1.Position[5].Pos := 183464;
   PRODUCT_TYPE[7].Motion.Ring_Turntable_Axis_1.Position[6].Pos := 228443;
   PRODUCT_TYPE[7].Motion.Ring_Turntable_Axis_1.Position[7].Pos := 273535;
   PRODUCT_TYPE[7].Motion.Ring_Turntable_Axis_1.Position[8].Pos := 318250;
   PRODUCT_TYPE[8].Motion.Ring_Turntable_Axis_1.Position[1].Pos := 3419;
   PRODUCT_TYPE[8].Motion.Ring_Turntable_Axis_1.Position[2].Pos := 48386;
   PRODUCT_TYPE[8].Motion.Ring_Turntable_Axis_1.Position[3].Pos := 93294;
   PRODUCT_TYPE[8].Motion.Ring_Turntable_Axis_1.Position[4].Pos := 138335;
   PRODUCT_TYPE[8].Motion.Ring_Turntable_Axis_1.Position[5].Pos := 183464;
   PRODUCT_TYPE[8].Motion.Ring_Turntable_Axis_1.Position[6].Pos := 228443;
   PRODUCT_TYPE[8].Motion.Ring_Turntable_Axis_1.Position[7].Pos := 273535;
   PRODUCT_TYPE[8].Motion.Ring_Turntable_Axis_1.Position[8].Pos := 318250;
   PRODUCT_TYPE[9].Motion.Ring_Turntable_Axis_1.Position[1].Pos := 3419;
   PRODUCT_TYPE[9].Motion.Ring_Turntable_Axis_1.Position[2].Pos := 48386;
   PRODUCT_TYPE[9].Motion.Ring_Turntable_Axis_1.Position[3].Pos := 93294;
   PRODUCT_TYPE[9].Motion.Ring_Turntable_Axis_1.Position[4].Pos := 138335;
   PRODUCT_TYPE[9].Motion.Ring_Turntable_Axis_1.Position[5].Pos := 183464;
   PRODUCT_TYPE[9].Motion.Ring_Turntable_Axis_1.Position[6].Pos := 228443;
   PRODUCT_TYPE[9].Motion.Ring_Turntable_Axis_1.Position[7].Pos := 273535;
   PRODUCT_TYPE[9].Motion.Ring_Turntable_Axis_1.Position[8].Pos := 318250;
   PRODUCT_TYPE[10].Motion.Ring_Turntable_Axis_1.Position[1].Pos := 3419;
   PRODUCT_TYPE[10].Motion.Ring_Turntable_Axis_1.Position[2].Pos := 48386;
   PRODUCT_TYPE[10].Motion.Ring_Turntable_Axis_1.Position[3].Pos := 93294;
   PRODUCT_TYPE[10].Motion.Ring_Turntable_Axis_1.Position[4].Pos := 138335;
   PRODUCT_TYPE[10].Motion.Ring_Turntable_Axis_1.Position[5].Pos := 183464;
   PRODUCT_TYPE[10].Motion.Ring_Turntable_Axis_1.Position[6].Pos := 228443;
   PRODUCT_TYPE[10].Motion.Ring_Turntable_Axis_1.Position[7].Pos := 273535;
   PRODUCT_TYPE[10].Motion.Ring_Turntable_Axis_1.Position[8].Pos := 318250;
   PRODUCT_TYPE[1].Motion.Ring_Turntable_Axis_1.Position[1..8].Vel := 10000;
   PRODUCT_TYPE[2].Motion.Ring_Turntable_Axis_1.Position[1..8].Vel := 10000;
   PRODUCT_TYPE[3].Motion.Ring_Turntable_Axis_1.Position[1..8].Vel := 10000;
   PRODUCT_TYPE[4].Motion.Ring_Turntable_Axis_1.Position[1..8].Vel := 10000;
   PRODUCT_TYPE[5].Motion.Ring_Turntable_Axis_1.Position[1..8].Vel := 10000;
   PRODUCT_TYPE[6].Motion.Ring_Turntable_Axis_1.Position[1..8].Vel := 10000;
   PRODUCT_TYPE[7].Motion.Ring_Turntable_Axis_1.Position[1..8].Vel := 10000;
   PRODUCT_TYPE[8].Motion.Ring_Turntable_Axis_1.Position[1..8].Vel := 10000;
   PRODUCT_TYPE[9].Motion.Ring_Turntable_Axis_1.Position[1..8].Vel := 10000;
   PRODUCT_TYPE[10].Motion.Ring_Turntable_Axis_1.Position[1..8].Vel := 10000;
   PRODUCT_TYPE[1].Motion.Shaft_Scan_Turntable_Axis.Position[2].Pos := 450000;
   PRODUCT_TYPE[1].Motion.Shaft_Scan_Turntable_Axis.Position[3].Pos := 900000;
   PRODUCT_TYPE[1].Motion.Shaft_Scan_Turntable_Axis.Position[4].Pos := 135000;
   PRODUCT_TYPE[1].Motion.Shaft_Scan_Turntable_Axis.Position[5].Pos := 180000;
   PRODUCT_TYPE[1].Motion.Shaft_Scan_Turntable_Axis.Position[6].Pos := 225000;
   PRODUCT_TYPE[1].Motion.Shaft_Scan_Turntable_Axis.Position[7].Pos := 270000;
   PRODUCT_TYPE[1].Motion.Shaft_Scan_Turntable_Axis.Position[8].Pos := 315000;
   PRODUCT_TYPE[2].Motion.Shaft_Scan_Turntable_Axis.Position[2].Pos := 450000;
   PRODUCT_TYPE[2].Motion.Shaft_Scan_Turntable_Axis.Position[3].Pos := 900000;
   PRODUCT_TYPE[2].Motion.Shaft_Scan_Turntable_Axis.Position[4].Pos := 135000;
   PRODUCT_TYPE[2].Motion.Shaft_Scan_Turntable_Axis.Position[5].Pos := 180000;
   PRODUCT_TYPE[2].Motion.Shaft_Scan_Turntable_Axis.Position[6].Pos := 225000;
   PRODUCT_TYPE[2].Motion.Shaft_Scan_Turntable_Axis.Position[7].Pos := 270000;
   PRODUCT_TYPE[2].Motion.Shaft_Scan_Turntable_Axis.Position[8].Pos := 315000;
   PRODUCT_TYPE[3].Motion.Shaft_Scan_Turntable_Axis.Position[2].Pos := 450000;
   PRODUCT_TYPE[3].Motion.Shaft_Scan_Turntable_Axis.Position[3].Pos := 900000;
   PRODUCT_TYPE[3].Motion.Shaft_Scan_Turntable_Axis.Position[4].Pos := 135000;
   PRODUCT_TYPE[3].Motion.Shaft_Scan_Turntable_Axis.Position[5].Pos := 180000;
   PRODUCT_TYPE[3].Motion.Shaft_Scan_Turntable_Axis.Position[6].Pos := 225000;
   PRODUCT_TYPE[3].Motion.Shaft_Scan_Turntable_Axis.Position[7].Pos := 270000;
   PRODUCT_TYPE[3].Motion.Shaft_Scan_Turntable_Axis.Position[8].Pos := 315000;
   PRODUCT_TYPE[4].Motion.Shaft_Scan_Turntable_Axis.Position[2].Pos := 450000;
   PRODUCT_TYPE[4].Motion.Shaft_Scan_Turntable_Axis.Position[3].Pos := 900000;
   PRODUCT_TYPE[4].Motion.Shaft_Scan_Turntable_Axis.Position[4].Pos := 135000;
   PRODUCT_TYPE[4].Motion.Shaft_Scan_Turntable_Axis.Position[5].Pos := 180000;
   PRODUCT_TYPE[4].Motion.Shaft_Scan_Turntable_Axis.Position[6].Pos := 225000;
   PRODUCT_TYPE[4].Motion.Shaft_Scan_Turntable_Axis.Position[7].Pos := 270000;
   PRODUCT_TYPE[4].Motion.Shaft_Scan_Turntable_Axis.Position[8].Pos := 315000;
   PRODUCT_TYPE[5].Motion.Shaft_Scan_Turntable_Axis.Position[2].Pos := 450000;
   PRODUCT_TYPE[5].Motion.Shaft_Scan_Turntable_Axis.Position[3].Pos := 900000;
   PRODUCT_TYPE[5].Motion.Shaft_Scan_Turntable_Axis.Position[4].Pos := 135000;
   PRODUCT_TYPE[5].Motion.Shaft_Scan_Turntable_Axis.Position[5].Pos := 180000;
   PRODUCT_TYPE[5].Motion.Shaft_Scan_Turntable_Axis.Position[6].Pos := 225000;
   PRODUCT_TYPE[5].Motion.Shaft_Scan_Turntable_Axis.Position[7].Pos := 270000;
   PRODUCT_TYPE[5].Motion.Shaft_Scan_Turntable_Axis.Position[8].Pos := 315000;
   PRODUCT_TYPE[6].Motion.Shaft_Scan_Turntable_Axis.Position[2].Pos := 450000;
   PRODUCT_TYPE[6].Motion.Shaft_Scan_Turntable_Axis.Position[3].Pos := 900000;
   PRODUCT_TYPE[6].Motion.Shaft_Scan_Turntable_Axis.Position[4].Pos := 135000;
   PRODUCT_TYPE[6].Motion.Shaft_Scan_Turntable_Axis.Position[5].Pos := 180000;
   PRODUCT_TYPE[6].Motion.Shaft_Scan_Turntable_Axis.Position[6].Pos := 225000;
   PRODUCT_TYPE[6].Motion.Shaft_Scan_Turntable_Axis.Position[7].Pos := 270000;
   PRODUCT_TYPE[6].Motion.Shaft_Scan_Turntable_Axis.Position[8].Pos := 315000;
   PRODUCT_TYPE[7].Motion.Shaft_Scan_Turntable_Axis.Position[2].Pos := 450000;
   PRODUCT_TYPE[7].Motion.Shaft_Scan_Turntable_Axis.Position[3].Pos := 900000;
   PRODUCT_TYPE[7].Motion.Shaft_Scan_Turntable_Axis.Position[4].Pos := 135000;
   PRODUCT_TYPE[7].Motion.Shaft_Scan_Turntable_Axis.Position[5].Pos := 180000;
   PRODUCT_TYPE[7].Motion.Shaft_Scan_Turntable_Axis.Position[6].Pos := 225000;
   PRODUCT_TYPE[7].Motion.Shaft_Scan_Turntable_Axis.Position[7].Pos := 270000;
   PRODUCT_TYPE[7].Motion.Shaft_Scan_Turntable_Axis.Position[8].Pos := 315000;
   PRODUCT_TYPE[8].Motion.Shaft_Scan_Turntable_Axis.Position[2].Pos := 450000;
   PRODUCT_TYPE[8].Motion.Shaft_Scan_Turntable_Axis.Position[3].Pos := 900000;
   PRODUCT_TYPE[8].Motion.Shaft_Scan_Turntable_Axis.Position[4].Pos := 135000;
   PRODUCT_TYPE[8].Motion.Shaft_Scan_Turntable_Axis.Position[5].Pos := 180000;
   PRODUCT_TYPE[8].Motion.Shaft_Scan_Turntable_Axis.Position[6].Pos := 225000;
   PRODUCT_TYPE[8].Motion.Shaft_Scan_Turntable_Axis.Position[7].Pos := 270000;
   PRODUCT_TYPE[8].Motion.Shaft_Scan_Turntable_Axis.Position[8].Pos := 315000;
   PRODUCT_TYPE[9].Motion.Shaft_Scan_Turntable_Axis.Position[2].Pos := 450000;
   PRODUCT_TYPE[9].Motion.Shaft_Scan_Turntable_Axis.Position[3].Pos := 900000;
   PRODUCT_TYPE[9].Motion.Shaft_Scan_Turntable_Axis.Position[4].Pos := 135000;
   PRODUCT_TYPE[9].Motion.Shaft_Scan_Turntable_Axis.Position[5].Pos := 180000;
   PRODUCT_TYPE[9].Motion.Shaft_Scan_Turntable_Axis.Position[6].Pos := 225000;
   PRODUCT_TYPE[9].Motion.Shaft_Scan_Turntable_Axis.Position[7].Pos := 270000;
   PRODUCT_TYPE[9].Motion.Shaft_Scan_Turntable_Axis.Position[8].Pos := 315000;
   PRODUCT_TYPE[10].Motion.Shaft_Scan_Turntable_Axis.Position[2].Pos := 450000;
   PRODUCT_TYPE[10].Motion.Shaft_Scan_Turntable_Axis.Position[3].Pos := 900000;
   PRODUCT_TYPE[10].Motion.Shaft_Scan_Turntable_Axis.Position[4].Pos := 135000;
   PRODUCT_TYPE[10].Motion.Shaft_Scan_Turntable_Axis.Position[5].Pos := 180000;
   PRODUCT_TYPE[10].Motion.Shaft_Scan_Turntable_Axis.Position[6].Pos := 225000;
   PRODUCT_TYPE[10].Motion.Shaft_Scan_Turntable_Axis.Position[7].Pos := 270000;
   PRODUCT_TYPE[10].Motion.Shaft_Scan_Turntable_Axis.Position[8].Pos := 315000;
   PRODUCT_TYPE[1].Motion.Shaft_Scan_Turntable_Axis.Position[1..8].Vel := 10000;
   PRODUCT_TYPE[2].Motion.Shaft_Scan_Turntable_Axis.Position[1..8].Vel := 10000;
   PRODUCT_TYPE[3].Motion.Shaft_Scan_Turntable_Axis.Position[1..8].Vel := 10000;
   PRODUCT_TYPE[4].Motion.Shaft_Scan_Turntable_Axis.Position[1..8].Vel := 10000;
   PRODUCT_TYPE[5].Motion.Shaft_Scan_Turntable_Axis.Position[1..8].Vel := 10000;
   PRODUCT_TYPE[6].Motion.Shaft_Scan_Turntable_Axis.Position[1..8].Vel := 10000;
   PRODUCT_TYPE[7].Motion.Shaft_Scan_Turntable_Axis.Position[1..8].Vel := 10000;
   PRODUCT_TYPE[8].Motion.Shaft_Scan_Turntable_Axis.Position[1..8].Vel := 10000;
   PRODUCT_TYPE[9].Motion.Shaft_Scan_Turntable_Axis.Position[1..8].Vel := 10000;
   PRODUCT_TYPE[10].Motion.Shaft_Scan_Turntable_Axis.Position[1..8].Vel := 10000;
   PRODUCT_TYPE[1].Motion.Gluing_Rotary_Jig_Axis.Position[3..6].Pos := 680000;
   PRODUCT_TYPE[1].Motion.Gluing_Rotary_Jig_Axis.Position[7].Pos := 90000;
   PRODUCT_TYPE[1].Motion.Gluing_Rotary_Jig_Axis.Position[8].Pos := 180000;
   PRODUCT_TYPE[1].Motion.Gluing_Rotary_Jig_Axis.Position[9].Pos := 270000;
   PRODUCT_TYPE[2].Motion.Gluing_Rotary_Jig_Axis.Position[3..6].Pos := 680000;
   PRODUCT_TYPE[2].Motion.Gluing_Rotary_Jig_Axis.Position[7].Pos := 90000;
   PRODUCT_TYPE[2].Motion.Gluing_Rotary_Jig_Axis.Position[8].Pos := 180000;
   PRODUCT_TYPE[2].Motion.Gluing_Rotary_Jig_Axis.Position[9].Pos := 270000;
   PRODUCT_TYPE[3].Motion.Gluing_Rotary_Jig_Axis.Position[3..6].Pos := 680000;
   PRODUCT_TYPE[3].Motion.Gluing_Rotary_Jig_Axis.Position[7].Pos := 90000;
   PRODUCT_TYPE[3].Motion.Gluing_Rotary_Jig_Axis.Position[8].Pos := 180000;
   PRODUCT_TYPE[3].Motion.Gluing_Rotary_Jig_Axis.Position[9].Pos := 270000;
   PRODUCT_TYPE[4].Motion.Gluing_Rotary_Jig_Axis.Position[3..6].Pos := 680000;
   PRODUCT_TYPE[4].Motion.Gluing_Rotary_Jig_Axis.Position[7].Pos := 90000;
   PRODUCT_TYPE[4].Motion.Gluing_Rotary_Jig_Axis.Position[8].Pos := 180000;
   PRODUCT_TYPE[4].Motion.Gluing_Rotary_Jig_Axis.Position[9].Pos := 270000;
   PRODUCT_TYPE[5].Motion.Gluing_Rotary_Jig_Axis.Position[3..6].Pos := 680000;
   PRODUCT_TYPE[5].Motion.Gluing_Rotary_Jig_Axis.Position[7].Pos := 90000;
   PRODUCT_TYPE[5].Motion.Gluing_Rotary_Jig_Axis.Position[8].Pos := 180000;
   PRODUCT_TYPE[5].Motion.Gluing_Rotary_Jig_Axis.Position[9].Pos := 270000;
   PRODUCT_TYPE[6].Motion.Gluing_Rotary_Jig_Axis.Position[3..6].Pos := 680000;
   PRODUCT_TYPE[6].Motion.Gluing_Rotary_Jig_Axis.Position[7].Pos := 90000;
   PRODUCT_TYPE[6].Motion.Gluing_Rotary_Jig_Axis.Position[8].Pos := 180000;
   PRODUCT_TYPE[6].Motion.Gluing_Rotary_Jig_Axis.Position[9].Pos := 270000;
   PRODUCT_TYPE[7].Motion.Gluing_Rotary_Jig_Axis.Position[3..6].Pos := 680000;
   PRODUCT_TYPE[7].Motion.Gluing_Rotary_Jig_Axis.Position[7].Pos := 90000;
   PRODUCT_TYPE[7].Motion.Gluing_Rotary_Jig_Axis.Position[8].Pos := 180000;
   PRODUCT_TYPE[7].Motion.Gluing_Rotary_Jig_Axis.Position[9].Pos := 270000;
   PRODUCT_TYPE[8].Motion.Gluing_Rotary_Jig_Axis.Position[3..6].Pos := 680000;
   PRODUCT_TYPE[8].Motion.Gluing_Rotary_Jig_Axis.Position[7].Pos := 90000;
   PRODUCT_TYPE[8].Motion.Gluing_Rotary_Jig_Axis.Position[8].Pos := 180000;
   PRODUCT_TYPE[8].Motion.Gluing_Rotary_Jig_Axis.Position[9].Pos := 270000;
   PRODUCT_TYPE[9].Motion.Gluing_Rotary_Jig_Axis.Position[3..6].Pos := 680000;
   PRODUCT_TYPE[9].Motion.Gluing_Rotary_Jig_Axis.Position[7].Pos := 90000;
   PRODUCT_TYPE[9].Motion.Gluing_Rotary_Jig_Axis.Position[8].Pos := 180000;
   PRODUCT_TYPE[9].Motion.Gluing_Rotary_Jig_Axis.Position[9].Pos := 270000;
   PRODUCT_TYPE[10].Motion.Gluing_Rotary_Jig_Axis.Position[3..6].Pos := 680000;
   PRODUCT_TYPE[10].Motion.Gluing_Rotary_Jig_Axis.Position[7].Pos := 90000;
   PRODUCT_TYPE[10].Motion.Gluing_Rotary_Jig_Axis.Position[8].Pos := 180000;
   PRODUCT_TYPE[10].Motion.Gluing_Rotary_Jig_Axis.Position[9].Pos := 270000;
   PRODUCT_TYPE[1].Motion.Gluing_Rotary_Jig_Axis.Position[1..2].Vel := 20000;
   PRODUCT_TYPE[1].Motion.Gluing_Rotary_Jig_Axis.Position[3..9].Vel := 10000;
   PRODUCT_TYPE[2].Motion.Gluing_Rotary_Jig_Axis.Position[1..2].Vel := 20000;
   PRODUCT_TYPE[2].Motion.Gluing_Rotary_Jig_Axis.Position[3..9].Vel := 10000;
   PRODUCT_TYPE[3].Motion.Gluing_Rotary_Jig_Axis.Position[1..2].Vel := 20000;
   PRODUCT_TYPE[3].Motion.Gluing_Rotary_Jig_Axis.Position[3..9].Vel := 10000;
   PRODUCT_TYPE[4].Motion.Gluing_Rotary_Jig_Axis.Position[1..2].Vel := 20000;
   PRODUCT_TYPE[4].Motion.Gluing_Rotary_Jig_Axis.Position[3..9].Vel := 10000;
   PRODUCT_TYPE[5].Motion.Gluing_Rotary_Jig_Axis.Position[1..2].Vel := 20000;
   PRODUCT_TYPE[5].Motion.Gluing_Rotary_Jig_Axis.Position[3..9].Vel := 10000;
   PRODUCT_TYPE[6].Motion.Gluing_Rotary_Jig_Axis.Position[1..2].Vel := 20000;
   PRODUCT_TYPE[6].Motion.Gluing_Rotary_Jig_Axis.Position[3..9].Vel := 10000;
   PRODUCT_TYPE[7].Motion.Gluing_Rotary_Jig_Axis.Position[1..2].Vel := 20000;
   PRODUCT_TYPE[7].Motion.Gluing_Rotary_Jig_Axis.Position[3..9].Vel := 10000;
   PRODUCT_TYPE[8].Motion.Gluing_Rotary_Jig_Axis.Position[1..2].Vel := 20000;
   PRODUCT_TYPE[8].Motion.Gluing_Rotary_Jig_Axis.Position[3..9].Vel := 10000;
   PRODUCT_TYPE[9].Motion.Gluing_Rotary_Jig_Axis.Position[1..2].Vel := 20000;
   PRODUCT_TYPE[9].Motion.Gluing_Rotary_Jig_Axis.Position[3..9].Vel := 10000;
   PRODUCT_TYPE[10].Motion.Gluing_Rotary_Jig_Axis.Position[1..2].Vel := 20000;
   PRODUCT_TYPE[10].Motion.Gluing_Rotary_Jig_Axis.Position[3..9].Vel := 10000;
   PRODUCT_TYPE[1].Motion.Ring_Turntable_Axis_2.Position[1].Pos := 3585;
   PRODUCT_TYPE[1].Motion.Ring_Turntable_Axis_2.Position[2].Pos := 48610;
   PRODUCT_TYPE[1].Motion.Ring_Turntable_Axis_2.Position[3].Pos := 93637;
   PRODUCT_TYPE[1].Motion.Ring_Turntable_Axis_2.Position[4].Pos := 138606;
   PRODUCT_TYPE[1].Motion.Ring_Turntable_Axis_2.Position[5].Pos := 183388;
   PRODUCT_TYPE[1].Motion.Ring_Turntable_Axis_2.Position[6].Pos := 228458;
   PRODUCT_TYPE[1].Motion.Ring_Turntable_Axis_2.Position[7].Pos := 273513;
   PRODUCT_TYPE[1].Motion.Ring_Turntable_Axis_2.Position[8].Pos := 318501;
   PRODUCT_TYPE[2].Motion.Ring_Turntable_Axis_2.Position[1].Pos := 3585;
   PRODUCT_TYPE[2].Motion.Ring_Turntable_Axis_2.Position[2].Pos := 48610;
   PRODUCT_TYPE[2].Motion.Ring_Turntable_Axis_2.Position[3].Pos := 93637;
   PRODUCT_TYPE[2].Motion.Ring_Turntable_Axis_2.Position[4].Pos := 138606;
   PRODUCT_TYPE[2].Motion.Ring_Turntable_Axis_2.Position[5].Pos := 183388;
   PRODUCT_TYPE[2].Motion.Ring_Turntable_Axis_2.Position[6].Pos := 228458;
   PRODUCT_TYPE[2].Motion.Ring_Turntable_Axis_2.Position[7].Pos := 273513;
   PRODUCT_TYPE[2].Motion.Ring_Turntable_Axis_2.Position[8].Pos := 318501;
   PRODUCT_TYPE[3].Motion.Ring_Turntable_Axis_2.Position[1].Pos := 3585;
   PRODUCT_TYPE[3].Motion.Ring_Turntable_Axis_2.Position[2].Pos := 48610;
   PRODUCT_TYPE[3].Motion.Ring_Turntable_Axis_2.Position[3].Pos := 93637;
   PRODUCT_TYPE[3].Motion.Ring_Turntable_Axis_2.Position[4].Pos := 138606;
   PRODUCT_TYPE[3].Motion.Ring_Turntable_Axis_2.Position[5].Pos := 183388;
   PRODUCT_TYPE[3].Motion.Ring_Turntable_Axis_2.Position[6].Pos := 228458;
   PRODUCT_TYPE[3].Motion.Ring_Turntable_Axis_2.Position[7].Pos := 273513;
   PRODUCT_TYPE[3].Motion.Ring_Turntable_Axis_2.Position[8].Pos := 318501;
   PRODUCT_TYPE[4].Motion.Ring_Turntable_Axis_2.Position[1].Pos := 3585;
   PRODUCT_TYPE[4].Motion.Ring_Turntable_Axis_2.Position[2].Pos := 48610;
   PRODUCT_TYPE[4].Motion.Ring_Turntable_Axis_2.Position[3].Pos := 93637;
   PRODUCT_TYPE[4].Motion.Ring_Turntable_Axis_2.Position[4].Pos := 138606;
   PRODUCT_TYPE[4].Motion.Ring_Turntable_Axis_2.Position[5].Pos := 183388;
   PRODUCT_TYPE[4].Motion.Ring_Turntable_Axis_2.Position[6].Pos := 228458;
   PRODUCT_TYPE[4].Motion.Ring_Turntable_Axis_2.Position[7].Pos := 273513;
   PRODUCT_TYPE[4].Motion.Ring_Turntable_Axis_2.Position[8].Pos := 318501;
   PRODUCT_TYPE[5].Motion.Ring_Turntable_Axis_2.Position[1].Pos := 3585;
   PRODUCT_TYPE[5].Motion.Ring_Turntable_Axis_2.Position[2].Pos := 48610;
   PRODUCT_TYPE[5].Motion.Ring_Turntable_Axis_2.Position[3].Pos := 93637;
   PRODUCT_TYPE[5].Motion.Ring_Turntable_Axis_2.Position[4].Pos := 138606;
   PRODUCT_TYPE[5].Motion.Ring_Turntable_Axis_2.Position[5].Pos := 183388;
   PRODUCT_TYPE[5].Motion.Ring_Turntable_Axis_2.Position[6].Pos := 228458;
   PRODUCT_TYPE[5].Motion.Ring_Turntable_Axis_2.Position[7].Pos := 273513;
   PRODUCT_TYPE[5].Motion.Ring_Turntable_Axis_2.Position[8].Pos := 318501;
   PRODUCT_TYPE[6].Motion.Ring_Turntable_Axis_2.Position[1].Pos := 3585;
   PRODUCT_TYPE[6].Motion.Ring_Turntable_Axis_2.Position[2].Pos := 48610;
   PRODUCT_TYPE[6].Motion.Ring_Turntable_Axis_2.Position[3].Pos := 93637;
   PRODUCT_TYPE[6].Motion.Ring_Turntable_Axis_2.Position[4].Pos := 138606;
   PRODUCT_TYPE[6].Motion.Ring_Turntable_Axis_2.Position[5].Pos := 183388;
   PRODUCT_TYPE[6].Motion.Ring_Turntable_Axis_2.Position[6].Pos := 228458;
   PRODUCT_TYPE[6].Motion.Ring_Turntable_Axis_2.Position[7].Pos := 273513;
   PRODUCT_TYPE[6].Motion.Ring_Turntable_Axis_2.Position[8].Pos := 318501;
   PRODUCT_TYPE[7].Motion.Ring_Turntable_Axis_2.Position[1].Pos := 3585;
   PRODUCT_TYPE[7].Motion.Ring_Turntable_Axis_2.Position[2].Pos := 48610;
   PRODUCT_TYPE[7].Motion.Ring_Turntable_Axis_2.Position[3].Pos := 93637;
   PRODUCT_TYPE[7].Motion.Ring_Turntable_Axis_2.Position[4].Pos := 138606;
   PRODUCT_TYPE[7].Motion.Ring_Turntable_Axis_2.Position[5].Pos := 183388;
   PRODUCT_TYPE[7].Motion.Ring_Turntable_Axis_2.Position[6].Pos := 228458;
   PRODUCT_TYPE[7].Motion.Ring_Turntable_Axis_2.Position[7].Pos := 273513;
   PRODUCT_TYPE[7].Motion.Ring_Turntable_Axis_2.Position[8].Pos := 318501;
   PRODUCT_TYPE[8].Motion.Ring_Turntable_Axis_2.Position[1].Pos := 3585;
   PRODUCT_TYPE[8].Motion.Ring_Turntable_Axis_2.Position[2].Pos := 48610;
   PRODUCT_TYPE[8].Motion.Ring_Turntable_Axis_2.Position[3].Pos := 93637;
   PRODUCT_TYPE[8].Motion.Ring_Turntable_Axis_2.Position[4].Pos := 138606;
   PRODUCT_TYPE[8].Motion.Ring_Turntable_Axis_2.Position[5].Pos := 183388;
   PRODUCT_TYPE[8].Motion.Ring_Turntable_Axis_2.Position[6].Pos := 228458;
   PRODUCT_TYPE[8].Motion.Ring_Turntable_Axis_2.Position[7].Pos := 273513;
   PRODUCT_TYPE[8].Motion.Ring_Turntable_Axis_2.Position[8].Pos := 318501;
   PRODUCT_TYPE[9].Motion.Ring_Turntable_Axis_2.Position[1].Pos := 3585;
   PRODUCT_TYPE[9].Motion.Ring_Turntable_Axis_2.Position[2].Pos := 48610;
   PRODUCT_TYPE[9].Motion.Ring_Turntable_Axis_2.Position[3].Pos := 93637;
   PRODUCT_TYPE[9].Motion.Ring_Turntable_Axis_2.Position[4].Pos := 138606;
   PRODUCT_TYPE[9].Motion.Ring_Turntable_Axis_2.Position[5].Pos := 183388;
   PRODUCT_TYPE[9].Motion.Ring_Turntable_Axis_2.Position[6].Pos := 228458;
   PRODUCT_TYPE[9].Motion.Ring_Turntable_Axis_2.Position[7].Pos := 273513;
   PRODUCT_TYPE[9].Motion.Ring_Turntable_Axis_2.Position[8].Pos := 318501;
   PRODUCT_TYPE[10].Motion.Ring_Turntable_Axis_2.Position[1].Pos := 3585;
   PRODUCT_TYPE[10].Motion.Ring_Turntable_Axis_2.Position[2].Pos := 48610;
   PRODUCT_TYPE[10].Motion.Ring_Turntable_Axis_2.Position[3].Pos := 93637;
   PRODUCT_TYPE[10].Motion.Ring_Turntable_Axis_2.Position[4].Pos := 138606;
   PRODUCT_TYPE[10].Motion.Ring_Turntable_Axis_2.Position[5].Pos := 183388;
   PRODUCT_TYPE[10].Motion.Ring_Turntable_Axis_2.Position[6].Pos := 228458;
   PRODUCT_TYPE[10].Motion.Ring_Turntable_Axis_2.Position[7].Pos := 273513;
   PRODUCT_TYPE[10].Motion.Ring_Turntable_Axis_2.Position[8].Pos := 318501;
   PRODUCT_TYPE[1].Motion.Ring_Turntable_Axis_2.Position[1..8].Vel := 10000;
   PRODUCT_TYPE[2].Motion.Ring_Turntable_Axis_2.Position[1..8].Vel := 10000;
   PRODUCT_TYPE[3].Motion.Ring_Turntable_Axis_2.Position[1..8].Vel := 10000;
   PRODUCT_TYPE[4].Motion.Ring_Turntable_Axis_2.Position[1..8].Vel := 10000;
   PRODUCT_TYPE[5].Motion.Ring_Turntable_Axis_2.Position[1..8].Vel := 10000;
   PRODUCT_TYPE[6].Motion.Ring_Turntable_Axis_2.Position[1..8].Vel := 10000;
   PRODUCT_TYPE[7].Motion.Ring_Turntable_Axis_2.Position[1..8].Vel := 10000;
   PRODUCT_TYPE[8].Motion.Ring_Turntable_Axis_2.Position[1..8].Vel := 10000;
   PRODUCT_TYPE[9].Motion.Ring_Turntable_Axis_2.Position[1..8].Vel := 10000;
   PRODUCT_TYPE[10].Motion.Ring_Turntable_Axis_2.Position[1..8].Vel := 10000;
END_DATA_BLOCK

DATA_BLOCK "DB_PARAMETERS_TEACH"   // DB7
{ S7_Optimized_Access := 'TRUE' }
// stored: MemoryReserve 100
   VAR
      HMI_PAGE_CONTROL : Struct
         TEACH_MODE_ACTIVE : Bool := FALSE;
         READ_CHOOSED_RECIPE : Bool := FALSE;
         NUMBER_OF_RECIPE : USInt := 1;
         SAVE_CHANGES_IN_RECIPE : Bool := FALSE;
         Use_recipe_Nbr : USInt := 1;
         Use_recipe_trigger : Bool := false;
         Speeds : Struct
            Glue_IAI : Struct
               X : Int := 10;
               Y : Int := 10;
               Z : Int := 10;
            END_STRUCT;
            A1_table : Int := 500;
            A2_table : Int := 500;
            Shaft_rotation : Int := 500;
            Glue_rotation : Int := 500;
         END_STRUCT;
         Go_to_pos : Struct
            Glue_IAI : Struct
               X : Real;
               Y : Real;
               Z : Real;
            END_STRUCT;
            A1_table : Int;
            A2_table : Int;
            Shaft_rotation : Int;
            Glue_rotation : Int;
         END_STRUCT;
         Go_to_pos_TRIGGER : Struct
            Glue_IAI : Struct
               X : Bool := FALSE;
               Y : Bool := FALSE;
               Z : Bool := FALSE;
            END_STRUCT;
            A1_table : Bool := FALSE;
            A2_table : Bool := FALSE;
            Shaft_rotation : Bool := FALSE;
            Glue_rotation : Bool := FALSE;
         END_STRUCT;
      END_STRUCT;
      "TEACH SCREEN VALUES" : "UDT_OP10_Recipe_type";
   END_VAR
BEGIN
END_DATA_BLOCK

DATA_BLOCK "DiagnosticDataBlock"   // DB3001
{ S7_Optimized_Access := 'FALSE' }
// stored: AutoNumber false
   VAR RETAIN
      DP : Struct
         DPReadStatus : Int;
         Status : Array[0..1023] of Bool;
      END_STRUCT;
      Profinet : Struct
         PNReadStatus : Int;
         Status : Array[0..1023] of Bool;
      END_STRUCT;
   END_VAR
BEGIN
   // DP.Status[0] : PLC-CPU
   // DP.Status[1] : Remote IO/ET200SP
   // DP.Status[2] : Festo Bus Coupler/总线耦合器
   // DP.Status[3] : CC-LINK
   // DP.Status[4] : Keyence Safety PLC
   // DP.Status[5] : Robot
   // DP.Status[6] : Keyence Laszer
   // DP.Status[7] : Balluff RFID
   // Profinet.Status[0] : ST70&ST80.PLC_CPU
   // Profinet.Status[1] : ST70&ST80.RFID
   // Profinet.Status[2] : ST70.Valves
   // Profinet.Status[3] : ST80.FCPN
   // Profinet.Status[4] : ST70.FCPN
   // Profinet.Status[5] : ST70.Screw
   // Profinet.Status[6] : CMMT-AS
   // Profinet.Status[7] : ST80.Screw
   // Profinet.Status[8] : ST80.Valves
END_DATA_BLOCK

DATA_BLOCK "Sys"   // DB3000
{ S7_Optimized_Access := 'FALSE' }
// stored: AutoNumber false
   VAR RETAIN
      COM : Struct   // Common
         AlwaysOFF : Bool := FALSE;
         AlwaysON : Bool := TRUE;
         FlashTime100mS : Bool := TRUE;   // Hardware Clock Memory 0.1S
         FlashTime200mS : Bool := TRUE;   // Hardware Clock Memory 0.2S
         FlashTime500mS : Bool := FALSE;   // Hardware Clock Memory 0.5S
         FlashTime1S : Bool := FALSE;   // Hardware Clock Memory 1S
         FlashTime2S : Bool := TRUE;   // Hardware Clock Memory 2S
         SpareBit : Bool := FALSE;
         PLCRestarted : Bool := TRUE;
      END_STRUCT;
      SpareB1 : Array[0..7] of Byte;
      DateTime : Struct   // DBX10.0
         Set : Date_And_Time := DT#1990-01-01-00:00:00;
         Read : Date_And_Time := DT#2025-03-12-08:03:05.785;
         Trigger : Bool := FALSE;   // Set
         ReturnValueRead : Int := 0;
         ReturnValueSet : Int := 0;
      END_STRUCT;
      SpareB2 : Array[0..17] of Byte;
      ScanTime : Struct   // DBX50.0
         CyclePrevious : Int := 14;
         CycleMax : Int := 23;
         CycleMin : Int := 9;
      END_STRUCT;
      RETVALI : Int := 0;
      RETVALW : Word := 16#0000;
      VersionManagement : Struct
         ProductLineName : String := 'Assembly Line';
         ProjectNumber : String[20] := 'SZ23055';
         "PLC IP Addr" : Array[0..3] of UInt;
         "HMI IP Addr" : Array[0..3] of UInt;
         PLCVersion : Array[0..1] of UInt;
         HMIVersion : Array[0..1] of UInt;
         "TIA Version" : String := 'TIA V18';
         StationID : Int := 10;
         HMIPageID : Int := 0;
      END_STRUCT;
   END_VAR
BEGIN
   SpareB1[0..7] := 16#00;
   SpareB2[0..17] := 16#00;
   VersionManagement."PLC IP Addr"[0] := 192;
   VersionManagement."PLC IP Addr"[1] := 168;
   VersionManagement."PLC IP Addr"[2..3] := 10;
   VersionManagement."HMI IP Addr"[0] := 192;
   VersionManagement."HMI IP Addr"[1] := 168;
   VersionManagement."HMI IP Addr"[2] := 45;
   VersionManagement."HMI IP Addr"[3] := 11;
   VersionManagement.PLCVersion[0] := 1;
   VersionManagement.PLCVersion[1] := 0;
   VersionManagement.HMIVersion[0] := 1;
   VersionManagement.HMIVersion[1] := 0;
END_DATA_BLOCK

DATA_BLOCK "ST10_GeneralData"   // DB1059
{ S7_Optimized_Access := 'FALSE' }
// stored: AutoNumber false
   VAR
      P_Plus : Array[0..50] of Bool;   // 脉冲沿信号使用Bool,使用需加注释
      ByPass : Array[0..10] of Bool;   // 屏蔽信号,使用需加注释
      HMI : Struct
         AREAPOINTER : Struct
            COORDINATION : Array[1..16] of Bool;
            USER_VERSION : Word;
            SCREEN_NUMBER : Struct
               SCREENTYPE : Int;
               SCREENNUMBER : Int;
               SPARE_1 : Int;
               FIELDNUMBER : Int;
               SPARE_2 : Int;
            END_STRUCT;
            JOB_MAILBOX : Struct
               JOBNUMBER : Int;
               PARAMETER_1 : Int;
               PARAMETER_2 : Int;
               PARAMETER_3 : Int;
            END_STRUCT;
            DATE_TIME_OP : Array[1..12] of Byte;
            DATE_TIME_PLC : Array[1..12] of Byte;
            SPARE : Array[1..22] of Byte;
            DataRecord : Struct   // 数据记录
               RecipeNummer : Word;
               DataRecordNummer : Word;
               Reserve : Word;
               TransferStatus : Word;   // 0,允许传送；2正在传送；4传送已完成，没有错误；12传送完成，出现错误
               Reserve_1 : Word;
            END_STRUCT;
         END_STRUCT;
         Win : Struct   // 弹窗相关变量
            Win : Int;
            WinBullfer : Int;
            "10x弹窗" : Array[1..10] of Int;
            "20x弹窗" : Array[1..10] of Int;
            "30x弹窗" : Array[1..10] of Int;
            "40x弹窗" : Array[1..10] of Int;
            TON : Array[1..40] of TON_TIME;
            "INT" { S7_SetPoint := 'True'} : Array[1..40] of Int;
            "Bool" : Array[1..40] of Bool;
         END_STRUCT;
         StationLightPB : Bool;   // 设备照明按钮
      END_STRUCT;
      Operator : Struct   // 操作员信息
         "Name" : String;   // 姓名
         ID : String;   // 工号
      END_STRUCT;
      TowerLamp : Struct
         PreReady : Bool;   // 等待托盘/等待人工操作
         PreStart : Bool;   // 人工操作完成（自动站False）
         ProcessingFinish : Bool;   // 加工完了 （单个产品加工完成）下个循环开始复位
         Maintenance : Bool;   // 维护提示（缺料OR保养置位1） 无---Flase
      END_STRUCT;
      FlowPartStatus { S7_SetPoint := 'True'} : Array[1..32] of Int;
      FunctionDeSelect : Struct   // 功能屏蔽选择
         "A" : Struct   // 单站屏蔽
            DeSelectPB_Servo380A1 : Bool;
            FunctionDeSelected_Servo380A1 : Bool;
            DeSelectPB_Servo381A1 : Bool;
            FunctionDeSelected_Servo381A1 : Bool;
            DeSelectPB_Servo383A1 : Bool;
            FunctionDeSelected_Servo383A1 : Bool;
            DeSelectPB_Reader800A1 : Bool;
            FunctionDeSelected_Reader800A1 : Bool;
            DeSelectPB_Reader801A1 : Bool;
            FunctionDeSelected_Reader801A1 : Bool;
            DeSelectPB_Reader802A1 : Bool;
            FunctionDeSelected_Reader802A1 : Bool;
            DeSelectPB_Reader803A1 : Bool;
            FunctionDeSelected_Reader803A1 : Bool;
            DeSelectPB_Reader804A1 : Bool;
            FunctionDeSelected_Reader804A1 : Bool;
         END_STRUCT;
         "B" : Struct   // RFID屏蔽
            DeSelectPB_Press372A1 : Bool;
            FunctionDeSelected_Press372A1 : Bool;
            DeSelectPB_Press375A1 : Bool;
            FunctionDeSelected_Press375A1 : Bool;
            DeSelectPB_Reader806A1 : Bool;
            FunctionDeSelected_Reader806A1 : Bool;
            DeSelectPB_TestPress372A1 : Bool;
            FunctionDeSelected_TestPress372A1 : Bool;
            DeSelectPB_TestPress375A1 : Bool;
            FunctionDeSelected_TestPress375A1 : Bool;
         END_STRUCT;
         C : Struct   // 扫码枪屏蔽
            DeSelectPB_Servo382A1 : Bool;
            FunctionDeSelected_Servo382A1 : Bool;
            DeSelectPB_ServoIAI : Bool;
            FunctionDeSelected_ServoIAI : Bool;
            DeSelectPB_IV3810A1 : Bool;
            FunctionDeSelected_IV3810A1 : Bool;
            DeSelectPB_IV3811A1 : Bool;
            FunctionDeSelected_IV3811A1 : Bool;
            DeSelectPB_Glue : Bool;
            FunctionDeSelected_Glue : Bool;
         END_STRUCT;
         "E" : Struct   // 注油屏蔽
            DeSelectPB : Bool;
            FunctionDeSelected : Bool;
         END_STRUCT;
         F : Struct   // 螺丝枪屏蔽
            DeSelectPB_Reader805A1 : Bool;
            FunctionDeSelected_Reader805A1 : Bool;
         END_STRUCT;
         H : Struct   // 油漆笔屏蔽
            DeSelectPB : Bool;
            FunctionDeSelected : Bool;
         END_STRUCT;
         J : Struct   // 油漆笔屏蔽
            DeSelectPB : Bool;
            FunctionDeSelected : Bool;
         END_STRUCT;
         K : Struct   // 油漆笔屏蔽
            DeSelectPB : Bool;
            FunctionDeSelected : Bool;
         END_STRUCT;
         L : Struct   // 油漆笔屏蔽
            DeSelectPB : Bool;
            FunctionDeSelected : Bool;
         END_STRUCT;
         MES : Struct   // MES屏蔽
            DeSelectPB : Bool;
            FunctionDeSelected : Bool;
         END_STRUCT;
         Global : Struct
            DeSelectPB_DryMode : Bool;
            FunctionDeSelected_DryMode : Bool;
            DeSelectPB_ScanFixture : Bool;
            FunctionDeSelected_ScanFixture : Bool;
            Spare_2 : Bool;
            Spare_3 : Bool;
            Spare_4 : Bool;
            Spare_5 : Bool;
            Spare_6 : Bool;
            Spare_7 : Bool;
            Spare_8 : Bool;
            Spare_9 : Bool;
            Spare_10 : Bool;
            Spare_11 : Bool;
            Spare_12 : Bool;
            Spare_13 : Bool;
         END_STRUCT;
      END_STRUCT;
      FlowControl_Handshake : Array[1..32] of Struct   // 流程控制的互锁
         PartPresent : Bool;
         initi : Bool;   // 初始化
         Start : Bool;
         Running : Bool;
         Done : Bool;
         Bypass : Bool;
      END_STRUCT;
      FixtureIDCheck { S7_SetPoint := 'True'} : Array[1..16] of "FixtureCheck_UDT";   // 工装匹配
      ProcessData { S7_SetPoint := 'True'} : Array[0..5] of "ProcessDatad";
   END_VAR
BEGIN
   // FlowControl_Handshake[2].Bypass : 流程NG
   // FlowControl_Handshake[1] : 主加工流程控制的互锁
   // FlowControl_Handshake[2] : 打标流程控制的互锁
   // FlowControl_Handshake[3] : 产品定位流程控制的互锁
   // FlowControl_Handshake[4] : 贴标流程控制互锁
END_DATA_BLOCK

DATA_BLOCK "Station_Sys"   // DB1060
TITLE = Station system DB
{ S7_Optimized_Access := 'FALSE' }
AUTHOR : RCS
FAMILY : Sys
VERSION : 2.0
// update 20160218
// stored: AutoNumber false
   VAR RETAIN
      ScreenNo : Int;   // For change HMI screen
      SpareB01 : Array[0..7] of Byte;   // *******************************************************************************
      Status : "RCS_SysStatus_V1";   // DBX10.0
      Input : Struct   // DBX20.0 For change PLC I input to PLC inside bit
         OP1 : Struct
            "Function 1" : Bool;
            "Function 2" : Bool;
            "Function 3" : Bool;
            "Function 4" : Bool;
            "Function 5" : Bool;
            "Function 6" : Bool;
            "Function 7" : Bool;
            "Function 8" : Bool;
         END_STRUCT;
         OP2 : Struct
            "Function 1" : Bool;
            "Function 2" : Bool;
            "Function 3" : Bool;
         END_STRUCT;
         OP3 : Struct
            "Function 1" : Bool;
            "Function 2" : Bool;
            "Function 3" : Bool;
         END_STRUCT;
      END_STRUCT;
      SpareB02 : Array[0..13] of Byte;   // *******************************************************************************
      HMI : Struct   // DBX40.0 HMI relation
         AP : Struct   // Area Pointer struct
            S1 : Int;
            CurrentScreenID : Int;
            S3 : Int;
            S4 : Int;
            S5 : Int;
         END_STRUCT;
      END_STRUCT;
      Cmd : "RCS_SysCmd_V1";   // DBX50.0
      SpareB03 : Array[0..7] of Byte;   // *******************************************************************************
      Interface : "RCS_SysComInterface_V1";   // DBX60.0
      SpareB04 : Array[0..3] of Byte;   // *******************************************************************************
      Initial : Struct   // DBX70.0
         Set : Bool;   // Trigger by HMI Button,[0]Total trigger
         Running : Bool;   // [0]Total initial Running
         OK : Bool;   // finish
      END_STRUCT;
      SpareB05 : Array[0..27] of Byte;   // *******************************************************************************
      Auto : "RCS_SysAuto_V1";   // DBX100.0
      SpareB10 : Array[0..5] of Byte;   // *******************************************************************************
      "A" : Struct   // DBX110.0 Auto control bit for some device
         "Device1 Auto control" : Bool;
         "Device2 Auto control" : Bool;
         "Device3 Auto control" : Bool;
         "Device4 Auto control" : Bool;
         "Device 01" : Struct
            "Function 1" : Bool;   // Flash
            "Function 2" : Bool;
            "Function 3" : Bool;   // Flash
         END_STRUCT;
         "Device 02" : Struct
            "Function 1" : Bool;   // Flash
            "Function 2" : Bool;
            "Function 3" : Bool;   // Flash
         END_STRUCT;
      END_STRUCT;
      SpareB11 : Array[0..33] of Byte;   // *******************************************************************************
      Manual : "RCS_SysManual_V1";   // DBX150.0
      SpareB12 : Array[0..6] of Byte;   // *******************************************************************************
      "M" : Struct   // DBX160.0 Manual control bit for some device
         "Device1 Manual control" : Bool;
         "Device2 Manual control" : Bool;
         "Device3 Manual control" : Bool;
         "Device4 Manual control" : Bool;
      END_STRUCT;
      SpareB13 : Array[0..37] of Byte;   // *******************************************************************************
      Safety : "RCS_SysSafety_V1";   // DBX200.0
      SpareB20 : Array[0..9] of Byte;   // *******************************************************************************
      Signal : Struct   // DBX220.0
         MainPressureSwitch1 : Bool;
         MainPressureSwitch2 : Bool;
         MainPressureSwitch3 : Bool;
      END_STRUCT;
      SpareB21 : Array[0..36] of Byte;   // *******************************************************************************
      Flag : Struct   // DBX260.0
         Processstart : Bool;
         PeocessComplete : Bool;
         IndexTable : Struct
            Interlock : Bool;
            TableRunning : Bool;   // Complete cycle Running
            StopandPosition : Bool;
            PositionOK : Bool;
            PositionNG : Bool;
            FixtureOK : Bool;
            FixtureNG : Bool;
            InitialOK : Bool;
         END_STRUCT;
      END_STRUCT;
      SpareB22 : Array[0..5] of Byte;   // *******************************************************************************
      P : Struct   // Positive RLO Edge Detection:-(P)- DBX270
         Record : Bool;
         "Set index run" : Bool;
         initial : Array[0..7] of Bool;
      END_STRUCT;
      SpareB23 : Array[0..5] of Byte;   // *******************************************************************************
      N : Struct   // Negative RLO Edge Detection:-(N)- DBX280
         Spare : Bool;
      END_STRUCT;
      SpareB24 : Array[0..17] of Byte;   // *******************************************************************************
      Alarm : "RCS_SysAlarmWarning_V1";   // DBX300.0
      SpareB30 : Array[0..7] of Byte;   // *******************************************************************************
      Warning : "RCS_SysAlarmWarning_V1";   // DBX310.0 / DBX500.0
      SpareB31 : Array[0..7] of Byte;   // *******************************************************************************
      AlarmTimes : Struct   // DBX320 If a fault continue happened over Limit times, than Auto running will be stopped / If a fault continue happened over Limit_times，Auto running will be stopped
         ForceStop : Bool;   // DBX320.0 / DBX650.0
         Reset : Bool;
         Limit : Int;
      END_STRUCT;
      SpareB33 : Array[0..5] of Byte;   // *******************************************************************************
      AlarmWarning : Int;   // DBX330 1:Alarm 2:Warning / DBX660 1:Alarm 2:Warning
      SpareB34 : Array[0..17] of Byte;   // *******************************************************************************
      Count : "RCS_SysCount_V1";   // DBX350.0 / DBX700.0
      SpareB40 : Array[0..11] of Byte;   // *******************************************************************************
      TotalCycleTime : "RCS_SysCycleTime_V1";   // DBX500.0 / DBX850.0
      SpareB41 : Array[0..11] of Byte;   // *******************************************************************************
      MachineCycleTime : "RCS_SysCycleTime_V1";   // DBX600.0 / DBX950.0
      SpareB42 : Array[0..11] of Byte;   // *******************************************************************************
      UserName { S7_SetPoint := 'True'} : String[20];   // DBX700.0
   END_VAR
BEGIN
   // Cmd.Record : 记录
   // Cmd.BuzzerOn : 蜂鸣器 On
   Cmd.OnOffLine := TRUE;
END_DATA_BLOCK

DATA_BLOCK "ST10_SysInput"   // DB1001
{ S7_Optimized_Access := 'TRUE' }
// stored: AutoNumber false, MemoryReserve 100
   VAR
      HMI_Button : Struct
         ControlOn : Bool := false;   // HMI_上电按钮
         ControlOff : Bool;   // HMI_断电按钮
         MachineStart : Bool := false;   // HMI_设备启动按钮
         MachineStop : Bool := false;   // HMI_设备停止按钮
         ResetButton : Bool := false;   // HMI_复位按钮
         "Manual/Auto" : Bool := false;   // HMI_手/自动切换按钮
         SafetyGateUnlock : Bool := false;   // HMI_安全门解锁按钮
         "E-Stop" : Bool := false;   // HMI_急停
      END_STRUCT;
      Sys : Struct
         iCircuitBreakerOK1 : Bool;   // 电子断路器 OK
         iCircuitBreakerOK2 : Bool;
         iPressure : Bool;   // 气压监控
      END_STRUCT;
      "iE-StopPB" : Array[1..20] of Bool;   // 急停按钮PB
      iSafetyGatFeedBack : Array[1..20] of Bool;   // 安全门
      iSafetydoorLockingFeedBack : Array[1..20] of Bool;   // 安全门反馈
      iMaterieldoorLockingFeedBack : Array[1..20] of Bool;   // 安全门反馈
   END_VAR
BEGIN
END_DATA_BLOCK

DATA_BLOCK "ST10_SysOutput"   // DB1002
{ S7_Optimized_Access := 'TRUE' }
// stored: AutoNumber false, MemoryReserve 100
   VAR
      oTowerLight : Struct
         Red : Bool;
         Yellow : Bool;
         Green : Bool;
         Blue : Bool;
      END_STRUCT;
      HMIButtonLight : Struct
         ControlOn : Bool := false;   // HMI_上电按钮
         ControlOff : Bool;   // HMI_断电按钮
         MachineStart : Bool := false;   // HMI_设备启动按钮
         MachineStop : Bool := false;   // HMI_设备停止按钮
         ResetButton : Bool := false;   // HMI_复位按钮
         "Manual/Auto" : Bool := false;   // HMI_手/自动切换按钮
         SafetyGateUnlock : Bool := false;   // HMI_安全门解锁按钮
      END_STRUCT;
      BoxLight : Struct
         oMachineStartLight : Bool;   // 启动按钮PB
         oMachineStopLight : Bool;   // 停止按钮PB
         oResetLight : Bool;   // 复位按钮PB
         oSafetyGateUnlockLight : Bool;   // 安全门解锁按钮PB
      END_STRUCT;
      SafetyDoorCoil : Array[1..20] of Bool;
      MaterialDoorCoil : Array[1..20] of Bool;
   END_VAR
BEGIN
END_DATA_BLOCK

